(* CoDeSys 2.3.9.59 project: HUS2_AS01_20210128.pro *)
(* Libraries: TcIMX53.lib 21.11.13 13:46:16, TcSUPS_CX9020_U900.lib 4.12.14 20:06:22, STANDARD.LIB 5.6.98 12:03:02, TcBase.lib 14.5.09 12:14:08, TcBaseMath.lib 27.7.04 12:07:56, TcFloatPC.lib 17.3.20 10:16:00, TcHVAC.lib 3.11.16 15:14:26, TcIoFunctions.lib 27.1.17 18:22:22, TcMath.lib 23.9.04 15:15:30, TcPlcCoupler.lib 26.7.12 16:14:58, TcSystem.lib 7.6.16 11:01:22, TcUtilities.lib 3.2.16 17:08:58, TcModbusSrv.lib 11.11.16 10:29:02 *)

(* Task configuration *)
TASK Standard (PRIORITY := 1, INTERVAL := T#20ms);
	MAIN
END_TASK

(* Global variable list: xOvrigt/AcknowledgeFault *)
VAR_GLOBAL
(****************************************************************************************************)
	bReset_Global		AT %Q*:	BOOL;	(*Global reset flag - this flag is common in many programs*)
END_VAR

(* Global variable list: xOvrigt/CtrlVoltage *)
VAR_GLOBAL
	bWithoutMonitoring							:	BOOL:=TRUE;
(*
	bCtrlVoltage_24VAC1		AT%I*			:	BOOL;			(* 24Volt AC1 *)
	bCtrlVoltage_24VAC2		AT%I*			:	BOOL;			(* 24Volt AC2 *)
	bCtrlVoltage_24VAC3		AT%I*			:	BOOL;			(* 24Volt AC3 *)
	bCtrlVoltage_24VAC4		AT%I*			:	BOOL;			(* 24Volt AC4 *)
	bCtrlVoltage_24VAC5		AT%I*			:	BOOL;			(* 24Volt AC5 *)
	bCtrlVoltage_24VAC6		AT%I*			:	BOOL;			(* 24Volt AC6 *)
	bCtrlVoltage_24VAC7		AT%I*			:	BOOL;			(* 24Volt AC7 *)
	bCtrlVoltage_24VAC8		AT%I*			:	BOOL;			(* 24Volt AC8 *)

	bCtrlVoltage_24VDC1	  	AT%I*			:	BOOL;			(* 24Volt DC1 *)
	bCtrlVoltage_24VDC2	  	AT%I*			:	BOOL;			(* 24Volt DC2 *)
	bCtrlVoltage_24VDC3	  	AT%I*			:	BOOL;			(* 24Volt DC3 *)
	bCtrlVoltage_24VDC4	  	AT%I*			:	BOOL;			(* 24Volt DC4 *)
	bCtrlVoltage_24VDC5	  	AT%I*			:	BOOL;			(* 24Volt DC5 *)
	bCtrlVoltage_24VDC6	  	AT%I*			:	BOOL;			(* 24Volt DC6 *)
	bCtrlVoltage_24VDC7	  	AT%I*			:	BOOL;			(* 24Volt DC7 *)
	bCtrlVoltage_24VDC8	  	AT%I*			:	BOOL;			(* 24Volt DC8 *)

	bCtrlVoltage_230VAC1	  	AT%I*			:	BOOL;			(* 230Volt AC1 *)
	bCtrlVoltage_230VAC2		AT%I*			:	BOOL;			(* 230Volt AC2 *)
	bCtrlVoltage_230VAC3	  	AT%I*			:	BOOL;			(* 230Volt AC3 *)
	bCtrlVoltage_230VAC4	  	AT%I*			:	BOOL;			(* 230Volt AC4 *)
	bCtrlVoltage_230VAC5	  	AT%I*			:	BOOL;			(* 230Volt AC5 *)
	bCtrlVoltage_230VAC6	  	AT%I*			:	BOOL;			(* 230Volt AC6 *)
	bCtrlVoltage_230VAC7	  	AT%I*			:	BOOL;			(* 230Volt AC7 *)
	bCtrlVoltage_230VAC8	  	AT%I*			:	BOOL;			(* 230Volt AC8 *)
*)
END_VAR

(* Global variable list: xOvrigt/Globale_Variablen *)
VAR_GLOBAL
	bSetDefault_Global:		BOOL;	(*Global set default flag. This flag is common in many programs*)

END_VAR

(* Global variable list: xOvrigt/GVL *)
VAR_GLOBAL

	HUS2_VV1_GT11_BV	AT%MB3260	:REAL;	(*	HUS2_VV1_GT11_BV	AS01	GVL.HUS2_VV1_GT11_BV	REAL	-50	150	-50	150	°C	0.0	Börvärde framledningstemp tappvarmvatten			*)


END_VAR

(* Global variable list: HUS1/AS02/HUS1_AS02_IO_Hardvara *)
VAR_GLOBAL


										
	(* Digitala in, KL1488  *)									
	(*Kort1*)									
		AS02_Kort01_DI01				AT %I*			:BOOL;	
		AS02_Kort01_DI02				AT %I*			:BOOL;	
		AS02_Kort01_DI03				AT %I*			:BOOL;	
		AS02_Kort01_DI04				AT %I*			:BOOL;	
		AS02_Kort01_DI05				AT %I*			:BOOL;	
		AS02_Kort01_DI06				AT %I*			:BOOL;	
		AS02_Kort01_DI07				AT %I*			:BOOL;	
		AS02_Kort01_DI08				AT %I*			:BOOL;	
										
										
	(* Digitala in, KL1488  *)									
	(*Kort2*)									
		AS02_Kort02_DI01				AT %I*			:BOOL;	
		AS02_Kort02_DI02				AT %I*			:BOOL;	
		AS02_Kort02_DI03				AT %I*			:BOOL;	
		AS02_Kort02_DI04				AT %I*			:BOOL;	
		AS02_Kort02_DI05				AT %I*			:BOOL;	
		AS02_Kort02_DI06				AT %I*			:BOOL;	
		AS02_Kort02_DI07				AT %I*			:BOOL;	
		AS02_Kort02_DI08				AT %I*			:BOOL;	
										
										
	(* Digital Ut, KL2408 *)									
	(*Kort3*)									
		AS02_Kort03_DU01				AT %Q*			:BOOL;	
		AS02_Kort03_DU02				AT %Q*			:BOOL;	
		AS02_Kort03_DU03				AT %Q*			:BOOL;	
		AS02_Kort03_DU04				AT %Q*			:BOOL;	
		AS02_Kort03_DU05				AT %Q*			:BOOL;	
		AS02_Kort03_DU06				AT %Q*			:BOOL;	
		AS02_Kort03_DU07				AT %Q*			:BOOL;	
		AS02_Kort03_DU08				AT %Q*			:BOOL;	
										
										
(*	(* Analoga in, KL3208-0010, PT1000 *)									
	(*Kort5*)									
		AS02_Kort04_AI01								
		AS02_Kort04_AI02								
		AS02_Kort04_AI03								
		AS02_Kort04_AI04								
		AS02_Kort04_AI05								
		AS02_Kort04_AI06								
		AS02_Kort04_AI07								
		AS02_Kort04_AI08					*)			
										

	(* Analoga Ut, KL4408 *)									
	(*Kort5*)									
		AS02_Kort05_AU01				AT %Q*			:INT;	
		AS02_Kort05_AU02				AT %Q*			:INT;	
		AS02_Kort05_AU03				AT %Q*			:INT;	
		AS02_Kort05_AU04				AT %Q*			:INT;	
		AS02_Kort05_AU05				AT %Q*			:INT;	
		AS02_Kort05_AU06				AT %Q*			:INT;	
		AS02_Kort05_AU07				AT %Q*			:INT;	
		AS02_Kort05_AU08				AT %Q*			:INT;	
										
										
										

										
										


END_VAR

(* Global variable list: HUS1/AS02/HUS1_AS02_IO_Program *)
VAR_GLOBAL

					(*	Name	Device	Address	Data type	Rawmin	Rawmax	Engmin	Engmax	Unit	Format	Description	Alarmoptions	Trendoptions	*)	
	(* Digitala in, KL1488  *)																			
	(*Kort 1*)																			
		HUS1_AS02_FB01_L	AT%MX332.0	:BOOL;	(*	HUS1_AS02_FB01_L	AS01	GVL.HUS1_AS02_FB01_L	DIGITAL	0	0	0	0			Fasbrott/fel fasföljd	p:A		*)
		HUS1_AS02_JFB01_L	AT%MX332.1	:BOOL;	(*	HUS1_AS02_JFB01_L	AS01	GVL.HUS1_AS02_JFB01_L	DIGITAL	0	0	0	0			Jordfelsbrytare 	p:B		*)	
		HUS1_AS02_LR01_L	AT%MX332.2	:BOOL;	(*	HUS1_AS02_LR01_L	AS01	GVL.HUS1_AS02_LR01_L	DIGITAL	0	0	0	0			Utlöst dvärgbrytare 	p:B		*)	
		HUS1_AS02_FS01_L	AT%MX332.3	:BOOL;	(*	HUS1_AS02_FS01_L	AS01	GVL.HUS1_AS02_FS01_L	DIGITAL	0	0	0	0			Utlöst finsäkring	p:B		*)	
		HUS1_AS02_RESERV_DI_KORT01_CH05	AT%MX332.4	:BOOL;	(*											Reserv 			*)	
		HUS1_AS02_RESERV_DI_KORT01_CH06	AT%MX332.5	:BOOL;	(*											Reserv 			*)	
		HUS1_AS02_RESERV_DI_KORT01_CH07	AT%MX332.6	:BOOL;	(*											Reserv 			*)	
		HUS1_AS02_RESERV_DI_KORT01_CH08	AT%MX332.7	:BOOL;	(*											Reserv 			*)	
																				

	(* Digitala in, KL1488  *)																			
	(*Kort 2*)																			
		HUS1_VS20_PV01_L	AT%MX333.3	:BOOL;	(*														*)
		HUS1_FA101_FF01_LD	AT%MX333.1	:BOOL;	(*	HUS1_FA101_FF01_LD	AS01	HUS1_AS02_Program.HUS1_FA101_FF01_LD	DIGITAL	0	0	0	0			Driftfel frånluftsfläkt			*)	
		HUS1_FA102_FF01_LD	AT%MX333.2	:BOOL;	(*	HUS1_FA102_FF01_LD	AS01	HUS1_AS02_Program.HUS1_FA102_FF01_LD	DIGITAL	0	0	0	0			Driftfel frånluftsfläkt			*)	
		HUS1_VS20_PV01_IT	AT%MX333.0	:BOOL;	(*	HUS1_VS20_PV01_IT	AS01	HUS1_AS02_Program.HUS1_VS20_PV01_IT	DIGITAL	0	0	0	0			Driftindikering cirkulationspump			*)	
		HUS1_AS02_RESERV_DI_KORT02_CH05	AT%MX333.4	:BOOL;	(*											Reserv 			*)	
		HUS1_AS02_RESERV_DI_KORT02_CH06	AT%MX333.5	:BOOL;	(*											Reserv 			*)	
		HUS1_AS02_RESERV_DI_KORT02_CH07	AT%MX333.6	:BOOL;	(*											Reserv 			*)	
		HUS1_AS02_RESERV_DI_KORT02_CH08	AT%MX333.7	:BOOL;	(*											Reserv 			*)	


	(* Digital Ut, KL2408 *)																			
	(*Kort 3*)																			
		HUS1_AS02_SA01_M	AT%MX334.0	:BOOL;	(*											Summalarm AS01 			*)	
		HUS1_VS20_PV01_M	AT%MX334.1	:BOOL;	(*											Manöver			*)	
		HUS1_AS02_RESERV_DU_KORT03_CH03	AT%MX334.2	:BOOL;	(*											Reserv 			*)	
		HUS1_AS02_RESERV_DU_KORT03_CH04	AT%MX334.3	:BOOL;	(*											Reserv 			*)	
		HUS1_AS02_RESERV_DU_KORT03_CH05	AT%MX334.4	:BOOL;	(*											Reserv 			*)	
		HUS1_AS02_RESERV_DU_KORT03_CH06	AT%MX334.5	:BOOL;	(*											Reserv 			*)	
		HUS1_AS02_RESERV_DU_KORT03_CH07	AT%MX334.6	:BOOL;	(*											Reserv 			*)	
		HUS1_AS02_RESERV_DU_KORT03_CH08	AT%MX334.7	:BOOL;	(*											Reserv 			*)	
																				
																				
	(* Analoga in, KL3208-0010, PT1000  *)																			
	(*Kort 4*)																			
		HUS1_VS20_GT11_MV	AT%MB336	:REAL;	(*	HUS1_VS20_GT11_MV	AS01	GVL.HUS1_VS20_GT11_MV	REAL	-50	150	-50	150	°C	0.0	Mätvärde tilloppstemperatur			*)	
		HUS1_VS20_GT41_MV	AT%MB340	:REAL;	(*	HUS1_VS20_GT41_MV	AS01	GVL.HUS1_VS20_GT41_MV	REAL	-50	150	-50	150	°C	0.0	Mätvärde returtemperatur			*)	
		HUS1_FA101_GT51_MV	AT%MB344	:REAL;	(*	HUS1_FA101_GT51_MV	AS01	GVL.HUS1_FA101_GT51_MV	REAL	-50	150	-50	150	°C	0.0	Mätvärde frånluftstemperatur			*)	
		HUS1_FA102_GT51_MV	AT%MB348	:REAL;	(*	HUS1_FA102_GT51_MV	AS01	GVL.HUS1_FA102_GT51_MV	REAL	-50	150	-50	150	°C	0.0	Mätvärde frånluftstemperatur			*)	
		HUS1_AS02_RESERV_AI_KORT04_CH05	AT%MB352	:REAL;	(*											Reserv			*)	
		HUS1_AS02_RESERV_AI_KORT04_CH06	AT%MB356	:REAL;	(*											Reserv			*)	
		HUS1_AS02_RESERV_AI_KORT04_CH07	AT%MB360	:REAL;	(*											Reserv			*)	
		HUS1_AS02_RESERV_AI_KORT04_CH08	AT%MB364	:REAL;	(*											Reserv			*)	
																				
																				
	(* Analoga ut, KL4408  *)																			
	(*Kort 5*)																			
		HUS1_VS20_SV21_R	AT%MB368	:REAL;	(*	HUS1_VS20_SV21_R	AS01	GVL.HUS1_VS20_SV21_R	REAL	0	100	0	100	%		Styrsignal ventilställdon			*)	
		HUS1_FA101_FF01_R	AT%MB372	:REAL;	(*	HUS1_FA101_FF01_R	AS01	GVL.HUS1_FA101_FF01_R	REAL	0	100	0	100	%		Styrsignal frånluftsfläkt			*)	
		HUS1_FA102_FF01_R	AT%MB376	:REAL;	(*	HUS1_FA102_FF01_R	AS01	GVL.HUS1_FA102_FF01_R	REAL	0	100	0	100	%		Styrsignal frånluftsfläkt			*)	
		HUS1_AS02_RESERV_AU_KORT05_CH04	AT%MB380	:REAL;	(*											Reserv			*)	
		HUS1_AS02_RESERV_AU_KORT05_CH05	AT%MB384	:REAL;	(*											Reserv			*)	
		HUS1_AS02_RESERV_AU_KORT05_CH06	AT%MB388	:REAL;	(*											Reserv			*)	
		HUS1_AS02_RESERV_AU_KORT05_CH07	AT%MB392	:REAL;	(*											Reserv			*)	
		HUS1_AS02_RESERV_AU_KORT05_CH08	AT%MB396	:REAL;	(*											Reserv			*)	
																				
																				
																				
																				

END_VAR

(* Global variable list: HUS1/FA101, FA102/HUS1_FA101_102_INST *)
VAR_GLOBAL PERSISTENT

																			

					(*	Name	Device	Address	Data type	Rawmin	Rawmax	Engmin	Engmax	Unit	Format	Description	Alarmoptions	Trendoptions	*)
																			
		HUS1_FA101_SO1_MAN	AT%MB4600	:INT;	(*	HUS1_FA101_SO1_MAN	AS01	GVL.HUS1_FA101_SO1_MAN	INT	0	2	0	2			Manuell styrning system FA101. 0=Auto, 1=Manuell från, 2=Manuell till			*)
		HUS1_FA101_SO1_FLM	AT%MB4602	:INT;	(*	HUS1_FA101_SO1_FLM	AS01	GVL.HUS1_FA101_SO1_FLM	INT	0	3600	0	3600	Min		Larmfördröjning serviceomkopplare ej i läge AUTO			*)
																			
		HUS1_FA101_FF01_FLM	AT%MB4604	:INT;	(*	HUS1_FA101_FF01_FLM	AS01	GVL.HUS1_FA101_FF01_FLM	INT	0	3600	0	3600	Min		Larmfördröjning frånluftsfläkt ej i AUTO			*)
		HUS1_FA101_FF01_FLD	AT%MB4606	:INT;	(*	HUS1_FA101_FF01_FLD	AS01	GVL.HUS1_FA101_FF01_FLD	INT	0	120	0	120	Sek		Larmfördröjning driftfel frånluftsfläkt			*)
																			
		HUS1_FA101_FF01_MAN	AT%MB4608	:INT;	(*	HUS1_FA101_FF01_MAN	AS01	GVL.HUS1_FA101_FF01_MAN	INT	0	2	0	2			Manuell styrning frånluftsfläkt 0=Auto,1=Från,2=Till			*)
		HUS1_FA101_FF01_MAN1	AT%MB4610	:INT;	(*	HUS1_FA101_FF01_MAN	AS01	GVL.HUS1_FA101_FF01_MAN	INT	0	1	0	1			Manuell styrning styrsignal frånluftsfläkt 0=Auto,1=Till			*)
		HUS1_FA101_FF01_RMAN	AT%MB4612	:REAL;	(*	HUS1_FA101_FF01_RMAN	AS01	GVL.HUS1_FA101_FF01_RMAN	REAL	0	100	0	100	%		Manuell styrsignal frånluftsfläkt			*)
																			
		HUS1_FA101_GT51_STAG	AT%MB4616	:REAL;	(*	HUS1_FA101_GT51_STAG	AS01	GVL.HUS1_FA101_GT51_STAG	REAL	0	50	0	50	°C	0.0	Gränsvärde start forcering frånluftsfläkt			*)
		HUS1_FA101_GT51_STOG	AT%MB4620	:REAL;	(*	HUS1_FA101_GT51_STOG	AS01	GVL.HUS1_FA101_GT51_STOG	REAL	0	50	0	50	°C	0.0	Gränsvärde stopp forcering frånluftsfläkt			*)
																			
		HUS1_FA101_GT51_GVH	AT%MB4624	:REAL;	(*	HUS1_FA101_GT51_GVH	AS01	GVL.HUS1_FA101_GT51_GVH	REAL	0	50	0	50	°C	0.0	Gränsvärde hög temperatur			*)
		HUS1_FA101_GT51_FLG	AT%MB4628	:INT;	(*	HUS1_FA101_GT51_FLG	AS01	GVL.HUS1_FA101_GT51_FLG	INT	0	3600	0	3600	Min		Lamfördröjning hög temperatur			*)
																			
																			
		HUS1_FA101_GT51_KRV	AT%MB4636	:REAL;	(*	HUS1_FA101_GT51_KRV	AS01	GVL.HUS1_FA101_GT51_KRV	REAL	-10	10	-10	10	°C	0.0	Kalibreringsvärde frånluftsgivare			*)
																			
		HUS1_FA101_FF01_BV	AT%MB4640	:REAL;	(*	HUS1_FA101_FF01_BV	AS01	GVL.HUS1_FA101_FF01_BV	REAL	0	100	0	100	%		Grundflöde frånluftsfläkt			*)
		HUS1_FA101_FF01_BV1	AT%MB4644	:REAL;	(*	HUS1_FA101_FF01_BV1	AS01	GVL.HUS1_FA101_FF01_BV1	REAL	0	100	0	100	%		Forcerat flöde frånluftsfläkt			*)
																			
																			
																			
																			
																			
																			
		HUS1_FA102_SO1_MAN	AT%MB4660	:INT;	(*	HUS1_FA102_SO1_MAN	AS01	GVL.HUS1_FA102_SO1_MAN	INT	0	2	0	2			Manuell styrning system FA102. 0=Auto, 1=Manuell från, 2=Manuell till			*)
		HUS1_FA102_SO1_FLM	AT%MB4662	:INT;	(*	HUS1_FA102_SO1_FLM	AS01	GVL.HUS1_FA102_SO1_FLM	INT	0	3600	0	3600	Min		Larmfördröjning serviceomkopplare ej i läge AUTO			*)
																			
		HUS1_FA102_FF01_FLM	AT%MB4664	:INT;	(*	HUS1_FA102_FF01_FLM	AS01	GVL.HUS1_FA102_FF01_FLM	INT	0	3600	0	3600	Min		Larmfördröjning frånluftsfläkt ej i AUTO			*)
		HUS1_FA102_FF01_FLD	AT%MB4666	:INT;	(*	HUS1_FA102_FF01_FLD	AS01	GVL.HUS1_FA102_FF01_FLD	INT	0	120	0	120	Sek		Larmfördröjning driftfel frånluftsfläkt			*)
																			
		HUS1_FA102_FF01_MAN	AT%MB4668	:INT;	(*	HUS1_FA102_FF01_MAN	AS01	GVL.HUS1_FA102_FF01_MAN	INT	0	2	0	2			Manuell styrning frånluftsfläkt 0=Auto,1=Från,2=Till			*)
		HUS1_FA102_FF01_MAN1	AT%MB4670	:INT;	(*	HUS1_FA102_FF01_MAN	AS01	GVL.HUS1_FA102_FF01_MAN	INT	0	1	0	1			Manuell styrning styrsignal frånluftsfläkt 0=Auto,1=Till			*)
		HUS1_FA102_FF01_RMAN	AT%MB4672	:REAL;	(*	HUS1_FA102_FF01_RMAN	AS01	GVL.HUS1_FA102_FF01_RMAN	REAL	0	100	0	100	%		Manuell styrsignal frånluftsfläkt			*)
																			
		HUS1_FA102_GT51_STAG	AT%MB4676	:REAL;	(*	HUS1_FA102_GT51_STAG	AS01	GVL.HUS1_FA102_GT51_STAG	REAL	0	50	0	50	°C	0.0	Gränsvärde start forcering frånluftsfläkt			*)
		HUS1_FA102_GT51_STOG	AT%MB4680	:REAL;	(*	HUS1_FA102_GT51_STOG	AS01	GVL.HUS1_FA102_GT51_STOG	REAL	0	50	0	50	°C	0.0	Gränsvärde stopp forcering frånluftsfläkt			*)
																			
		HUS1_FA102_GT51_GVH	AT%MB4684	:REAL;	(*	HUS1_FA102_GT51_GVH	AS01	GVL.HUS1_FA102_GT51_GVH	REAL	0	50	0	50	°C	0.0	Gränsvärde hög temperatur			*)
		HUS1_FA102_GT51_FLG	AT%MB4688	:INT;	(*	HUS1_FA102_GT51_FLG	AS01	GVL.HUS1_FA102_GT51_FLG	INT	0	3600	0	3600	Min		Lamfördröjning hög temperatur			*)
																			
																			
		HUS1_FA102_GT51_KRV	AT%MB4696	:REAL;	(*	HUS1_FA102_GT51_KRV	AS01	GVL.HUS1_FA102_GT51_KRV	REAL	-10	10	-10	10	°C	0.0	Kalibreringsvärde frånluftsgivare			*)
																			
		HUS1_FA102_FF01_BV	AT%MB4700	:REAL;	(*	HUS1_FA102_FF01_BV	AS01	GVL.HUS1_FA102_FF01_BV	REAL	0	100	0	100	%		Grundflöde frånluftsfläkt			*)
		HUS1_FA102_FF01_BV1	AT%MB4704	:REAL;	(*	HUS1_FA102_FF01_BV1	AS01	GVL.HUS1_FA102_FF01_BV1	REAL	0	100	0	100	%		Forcerat flöde frånluftsfläkt			*)
																			
																			
																			
																			
																			
																			
																			
																			

																			


END_VAR
																
																

(* Global variable list: HUS1/FA101, FA102/HUS1_FA101_102_LARM *)
VAR_GLOBAL



																						
																						
	HUS1_FA101_SO1_LM	AT%MX4780.0	:BOOL; 	(*	HUS1_FA101_SO1_LM	AS01	GVL.HUS1_FA101_SO1_LM	DIGITAL	0	0	0	0			Serviceomkopplare ej i läge AUTO	p:C		*)				
	HUS1_FA101_FF01_LM	AT%MX4780.1	:BOOL; 	(*	HUS1_FA101_FF01_LM	AS01	GVL.HUS1_FA101_FF01_LM	DIGITAL	0	0	0	0			Frånluftsfläkt ej i AUTO	p:B		*)				
	HUS1_FA101_GT51_LG	AT%MX4780.2	:BOOL; 	(*	HUS1_FA101_GT51_LG	AS01	GVL.HUS1_FA101_GT51_LG	DIGITAL	0	0	0	0			Givarfel frånluftsgivare	p:B		*)				
	HUS1_FA101_GT51_LH	AT%MX4780.3	:BOOL; 	(*	HUS1_FA101_GT51_LH	AS01	GVL.HUS1_FA101_GT51_LH	DIGITAL	0	0	0	0			Hög temperatur	p:B		*)				
																						
	HUS1_FA101_FF01_ACK	AT%MX4781.0	:BOOL; 	(*	HUS1_FA101_FF01_ACK	AS01	GVL.HUS1_FA101_FF01_ACK	DIGITAL	0	0	0	0			Larmkvittens frånluftsfläkt			*)				
																						
																						
	HUS1_FA102_SO1_LM	AT%MX4782.0	:BOOL; 	(*	HUS1_FA102_SO1_LM	AS01	GVL.HUS1_FA102_SO1_LM	DIGITAL	0	0	0	0			Serviceomkopplare ej i läge AUTO	p:C		*)				
	HUS1_FA102_FF01_LM	AT%MX4782.1	:BOOL; 	(*	HUS1_FA102_FF01_LM	AS01	GVL.HUS1_FA102_FF01_LM	DIGITAL	0	0	0	0			Frånluftsfläkt ej i AUTO	p:B		*)				
	HUS1_FA102_GT51_LG	AT%MX4782.2	:BOOL; 	(*	HUS1_FA102_GT51_LG	AS01	GVL.HUS1_FA102_GT51_LG	DIGITAL	0	0	0	0			Givarfel frånluftsgivare	p:B		*)				
	HUS1_FA102_GT51_LH	AT%MX4782.3	:BOOL; 	(*	HUS1_FA102_GT51_LH	AS01	GVL.HUS1_FA102_GT51_LH	DIGITAL	0	0	0	0			Hög temperatur	p:B		*)				
																						
	HUS1_FA102_FF01_ACK	AT%MX4784.0	:BOOL; 	(*	HUS1_FA102_FF01_ACK	AS01	GVL.HUS1_FA102_FF01_ACK	DIGITAL	0	0	0	0			Larmkvittens frånluftsfläkt			*)				
																						
																						
																						
																						



END_VAR

(* Global variable list: HUS1/FA101, FA102/HUS1_FA101_102_OVRIGT *)
VAR_GLOBAL


																				
	HUS1_FA101_SO1_IH	AT%MX4900.0	:BOOL;	(*	HUS1_FA101_SO1_IH	AS01	GVL.HUS1_FA101_SO1_IH	DIGITAL	0	0	0	0			Serviceomkopplare ej i AUTO			*)		
	HUS1_FA101_SO1_IA	AT%MX4900.1	:BOOL;	(*	HUS1_FA101_SO1_IA	AS01	GVL.HUS1_FA101_SO1_IA	DIGITAL	0	0	0	0			Serviceomkopplare i läge AUTO			*)		
	HUS1_FA101_SO1_IF	AT%MX4900.2	:BOOL;	(*	HUS1_FA101_SO1_IF	AS01	GVL.HUS1_FA101_SO1_IF	DIGITAL	0	0	0	0			Serviceomkopplare i läge 0			*)		
	HUS1_FA101_SO1_IT	AT%MX4900.3	:BOOL;	(*	HUS1_FA101_SO1_IT	AS01	GVL.HUS1_FA101_SO1_IT	DIGITAL	0	0	0	0			Serviceomkopplare i läge HAND TILL			*)		
																				
	HUS1_FA101_FF01_IT	AT%MX4900.5	:BOOL;	(*	HUS1_FA101_FF01_IT	AS01	GVL.HUS1_FA101_FF01_IT	DIGITAL	0	0	0	0			Frånluftsfläkt indikering TILL			*)		
																				
																				
	HUS1_FA102_SO1_IH	AT%MX4901.0	:BOOL;	(*	HUS1_FA102_SO1_IH	AS01	GVL.HUS1_FA102_SO1_IH	DIGITAL	0	0	0	0			Serviceomkopplare ej i AUTO			*)		
	HUS1_FA102_SO1_IA	AT%MX4901.1	:BOOL;	(*	HUS1_FA102_SO1_IA	AS01	GVL.HUS1_FA102_SO1_IA	DIGITAL	0	0	0	0			Serviceomkopplare i läge AUTO			*)		
	HUS1_FA102_SO1_IF	AT%MX4901.2	:BOOL;	(*	HUS1_FA102_SO1_IF	AS01	GVL.HUS1_FA102_SO1_IF	DIGITAL	0	0	0	0			Serviceomkopplare i läge 0			*)		
	HUS1_FA102_SO1_IT	AT%MX4901.3	:BOOL;	(*	HUS1_FA102_SO1_IT	AS01	GVL.HUS1_FA102_SO1_IT	DIGITAL	0	0	0	0			Serviceomkopplare i läge HAND TILL			*)		
																				
	HUS1_FA102_FF01_IT	AT%MX4901.5	:BOOL;	(*	HUS1_FA102_FF01_IT	AS01	GVL.HUS1_FA102_FF01_IT	DIGITAL	0	0	0	0			Frånluftsfläkt indikering TILL			*)		
																				
																				
																				
																				



END_VAR

(* Global variable list: HUS1/VS20/HUS1_VS20_INST *)
VAR_GLOBAL PERSISTENT


																			
					(*	Name	Device	Address	Data type	Rawmin	Rawmax	Engmin	Engmax	Unit	Format	Description	Alarmoptions	Trendoptions	*)
																			
		HUS1_VS20_GT11_UX1	AT%MB4392	:REAL;	(*	HUS1_VS20_GT11_UX1	AS01	GVL.HUS1_VS20_GT11_UX1	REAL	-50	150	-50	150	°C	0.0	Utetemp. kompenserad kurva Brytpunkt X1			*)
		HUS1_VS20_GT11_UX2	AT%MB4396	:REAL;	(*	HUS1_VS20_GT11_UX2	AS01	GVL.HUS1_VS20_GT11_UX2	REAL	-50	150	-50	150	°C	0.0	Utetemp. kompenserad kurva Brytpunkt X2			*)
		HUS1_VS20_GT11_UX3	AT%MB4400	:REAL;	(*	HUS1_VS20_GT11_UX3	AS01	GVL.HUS1_VS20_GT11_UX3	REAL	-50	150	-50	150	°C	0.0	Utetemp. kompenserad kurva Brytpunkt X3			*)
		HUS1_VS20_GT11_UX4	AT%MB4404	:REAL;	(*	HUS1_VS20_GT11_UX4	AS01	GVL.HUS1_VS20_GT11_UX4	REAL	-50	150	-50	150	°C	0.0	Utetemp. kompenserad kurva Brytpunkt X4			*)
		HUS1_VS20_GT11_UX5	AT%MB4408	:REAL;	(*	HUS1_VS20_GT11_UX5	AS01	GVL.HUS1_VS20_GT11_UX5	REAL	-50	150	-50	150	°C	0.0	Utetemp. kompenserad kurva Brytpunkt X5			*)
		HUS1_VS20_GT11_UY1	AT%MB4412	:REAL;	(*	HUS1_VS20_GT11_UY1	AS01	GVL.HUS1_VS20_GT11_UY1	REAL	0	150	0	150	°C	0.0	Utetemp. kompenserad kurva Brytpunkt Y1			*)
		HUS1_VS20_GT11_UY2	AT%MB4416	:REAL;	(*	HUS1_VS20_GT11_UY2	AS01	GVL.HUS1_VS20_GT11_UY2	REAL	0	150	0	150	°C	0.0	Utetemp. kompenserad kurva Brytpunkt Y2			*)
		HUS1_VS20_GT11_UY3	AT%MB4420	:REAL;	(*	HUS1_VS20_GT11_UY3	AS01	GVL.HUS1_VS20_GT11_UY3	REAL	0	150	0	150	°C	0.0	Utetemp. kompenserad kurva Brytpunkt Y3			*)
		HUS1_VS20_GT11_UY4	AT%MB4424	:REAL;	(*	HUS1_VS20_GT11_UY4	AS01	GVL.HUS1_VS20_GT11_UY4	REAL	0	150	0	150	°C	0.0	Utetemp. kompenserad kurva Brytpunkt Y4			*)
		HUS1_VS20_GT11_UY5	AT%MB4428	:REAL;	(*	HUS1_VS20_GT11_UY5	AS01	GVL.HUS1_VS20_GT11_UY5	REAL	0	150	0	150	°C	0.0	Utetemp. kompenserad kurva Brytpunkt Y5			*)
		HUS1_VS20_GT11_UMIN	AT%MB4432	:REAL;	(*	HUS1_VS20_GT11_UMIN	AS01	GVL.HUS1_VS20_GT11_UMIN	REAL	0	150	0	150	°C	0.0	Utetemp. kompenserad kurva Min-begränsning			*)
		HUS1_VS20_GT11_UMAX	AT%MB4436	:REAL;	(*	HUS1_VS20_GT11_UMAX	AS01	GVL.HUS1_VS20_GT11_UMAX	REAL	0	150	0	150	°C	0.0	Utetemp. kompenserad kurva Max-begränsning			*)
																			
		HUS1_VS20_GT11_CP	AT%MB4440	:REAL;	(*	HUS1_VS20_GT11_CPV	AS01	GVL.HUS1_VS20_GT11_CP	REAL	0	10	0	10		0.0	P-parameter			*)
		HUS1_VS20_GT11_CI	AT%MB4444	:REAL;	(*	HUS1_VS20_GT11_CIV	AS01	GVL.HUS1_VS20_GT11_CI	REAL	0	900	0	900	Sek		I-Tid 			*)
		HUS1_VS20_GT11_CD	AT%MB4448	:REAL;	(*	HUS1_VS20_GT11_CDV	AS01	GVL.HUS1_VS20_GT11_CD	REAL	0	900	0	900	Sek		D-tid 			*)
		HUS1_VS20_GT11_CS	AT%MB4452	:REAL;	(*	HUS1_VS20_GT11_CSV	AS01	GVL.HUS1_VS20_GT11_CS	REAL	0	900	0	900	Sek		Samplingstid			*)
		HUS1_VS20_GT11_CZ	AT%MB4456	:REAL;	(*	HUS1_VS20_GT11_CZV	AS01	GVL.HUS1_VS20_GT11_CZ	REAL	-10	10	-10	10	°C	0.0	Dödband regulator			*)
																			
		HUS1_VS20_SO1_MAN	AT%MB4460	:INT;	(*	HUS1_VS20_SO1_MAN	AS01	GVL.HUS1_VS20_SO1_MAN	INT	0	2	0	2			Manuell styrning system VS20. 0=Auto, 1=Manuell från, 2=Manuell till			*)
		HUS1_VS20_PV01_MAN	AT%MB4462	:INT;	(*	HUS1_VS20_PV01_MAN	AS01	GVL.HUS1_VS20_PV01_MAN	INT	0	2	0	2			Manuell styrning crikulationspump 0=Auto,1=Från,2=Till			*)
		HUS1_VS20_SV21_MAN1	AT%MB4464	:INT;	(*	HUS1_VS20_SV21_MAN	AS01	GVL.HUS1_VS20_SV21_MAN	INT	0	1	0	1			Manuell styrning ventilställdon 0=Auto,1=Hand			*)
		HUS1_VS20_SV21_RMAN	AT%MB4468	:REAL;	(*	HUS1_VS20_SV21_RMAN	AS01	GVL.HUS1_VS20_SV21_RMAN	REAL	0	100	0	100	%		Manuell styrsignal ventilställdon			*)
																			
		HUS1_VS20_SO1_FLM	AT%MB4472	:INT;	(*	HUS1_VS20_SO1_FLM	AS01	GVL.HUS1_VS20_SO1_FLM	INT	0	3600	0	3600	Min		Larmfördröjning serviceomkopplare ej i läge AUTO			*)
		HUS1_VS20_PV01_FLM	AT%MB4474	:INT;	(*	HUS1_VS20_PV01_FLM	AS01	GVL.HUS1_VS20_PV01_FLM	INT	0	3600	0	3600	Min		Larmfördröjning cirkulationspump ej i AUTO			*)
		HUS1_VS20_SV21_FLM	AT%MB4476	:INT;	(*	HUS1_VS20_SV21_FLM	AS01	GVL.HUS1_VS20_SV21_FLM	INT	0	3600	0	3600	Min		Larmfördröjning ventilställdon ej i AUTO			*)
		HUS1_VS20_PV01_FLD	AT%MB4478	:INT;	(*	HUS1_VS20_PV01_FLD	AS01	GVL.HUS1_VS20_PV01_FLD	INT	0	120	0	120	Sek		Larmfördröjning driftfel cirkulationspump			*)
																			
		HUS1_VS20_GT11_GAVH	AT%MB4484	:REAL;	(*	HUS1_VS20_GT11_GAVH	AS01	GVL.HUS1_VS20_GT11_GAVH	REAL	-20	20	-20	20	°C	0.0	Gränsavvikelse hög framledningstemperatur			*)
		HUS1_VS20_GT11_GAVL	AT%MB4488	:REAL;	(*	HUS1_VS20_GT11_GAVL	AS01	GVL.HUS1_VS20_GT11_GAVL	REAL	-20	20	-20	20	°C	0.0	Gränsavvikelse låg framledningstemperatur			*)
		HUS1_VS20_GT11_FLAH	AT%MB4492	:INT;	(*	HUS1_VS20_GT11_FLAH	AS01	GVL.HUS1_VS20_GT11_FLAH	INT	0	3600	0	3600	Min		Larmfördröjning hög framledningstemperatur			*)
		HUS1_VS20_GT11_FLAL	AT%MB4494	:INT;	(*	HUS1_VS20_GT11_FLAL	AS01	GVL.HUS1_VS20_GT11_FLAL	INT	0	3600	0	3600	Min		Lamfördröjning låg framledningstemperatur			*)
																			
																			
																			
																			
																			
																			
																			
																			
																			
		HUS1_VS20_GT11_KRV	AT%MB4496	:REAL;	(*	HUS1_VS20_GT11_KRV	AS01	GVL.HUS1_VS20_GT11_KRV	REAL	-10	10	-10	10	°C	0.0	Kalibreringsvärde framledningsgivare			*)
		HUS1_VS20_GT41_KRV	AT%MB4500	:REAL;	(*	HUS1_VS20_GT41_KRV	AS01	GVL.HUS1_VS20_GT41_KRV	REAL	-10	10	-10	10	°C	0.0	Kalibreringsvärde returgivare			*)
																			
																			
																			
		HUS1_VS20_GT11_X1	AT%MB4504	:REAL;	(*	HUS1_VS20_GT11_X1	AS01	GVL.HUS1_VS20_GT11_X1	REAL	-50	150	-50	150	°C	0.0	Effektbegränsning kurva Brytpunkt X1			*)
		HUS1_VS20_GT11_X2	AT%MB4508	:REAL;	(*	HUS1_VS20_GT11_X2	AS01	GVL.HUS1_VS20_GT11_X2	REAL	-50	150	-50	150	°C	0.0	Effektbegränsning kurva Brytpunkt X2			*)
		HUS1_VS20_GT11_X3	AT%MB4512	:REAL;	(*	HUS1_VS20_GT11_X3	AS01	GVL.HUS1_VS20_GT11_X3	REAL	-50	150	-50	150	°C	0.0	Effektbegränsning kurva Brytpunkt X3			*)
		HUS1_VS20_GT11_X4	AT%MB4516	:REAL;	(*	HUS1_VS20_GT11_X4	AS01	GVL.HUS1_VS20_GT11_X4	REAL	-50	150	-50	150	°C	0.0	Effektbegränsning kurva Brytpunkt X4			*)
		HUS1_VS20_GT11_X5	AT%MB4520	:REAL;	(*	HUS1_VS20_GT11_X5	AS01	GVL.HUS1_VS20_GT11_X5	REAL	-50	150	-50	150	°C	0.0	Effektbegränsning kurva Brytpunkt X5			*)
		HUS1_VS20_GT11_Y1	AT%MB4524	:REAL;	(*	HUS1_VS20_GT11_Y1	AS01	GVL.HUS1_VS20_GT11_Y1	REAL	0	150	0	150	°C	0.0	Effektbegränsning kurva Brytpunkt Y1			*)
		HUS1_VS20_GT11_Y2	AT%MB4528	:REAL;	(*	HUS1_VS20_GT11_Y2	AS01	GVL.HUS1_VS20_GT11_Y2	REAL	0	150	0	150	°C	0.0	Effektbegränsning kurva Brytpunkt Y2			*)
		HUS1_VS20_GT11_Y3	AT%MB4532	:REAL;	(*	HUS1_VS20_GT11_Y3	AS01	GVL.HUS1_VS20_GT11_Y3	REAL	0	150	0	150	°C	0.0	Effektbegränsning kurva Brytpunkt Y3			*)
		HUS1_VS20_GT11_Y4	AT%MB4536	:REAL;	(*	HUS1_VS20_GT11_Y4	AS01	GVL.HUS1_VS20_GT11_Y4	REAL	0	150	0	150	°C	0.0	Effektbegränsning kurva Brytpunkt Y4			*)
		HUS1_VS20_GT11_Y5	AT%MB4540	:REAL;	(*	HUS1_VS20_GT11_Y5	AS01	GVL.HUS1_VS20_GT11_Y5	REAL	0	150	0	150	°C	0.0	Effektbegränsning kurva Brytpunkt Y5			*)
		HUS1_VS20_GT11_MIN	AT%MB4544	:REAL;	(*	HUS1_VS20_GT11_MIN	AS01	GVL.HUS1_VS20_GT11_MIN	REAL	0	150	0	150	°C	0.0	Effektbegränsning kurva Min-begränsning			*)
		HUS1_VS20_GT11_MAX	AT%MB4548	:REAL;	(*	HUS1_VS20_GT11_MAX	AS01	GVL.HUS1_VS20_GT11_MAX	REAL	0	150	0	150	°C	0.0	Effektbegränsning kurva Max-begränsning			*)
																			
																			
																			
																			
																			
																			
																			



END_VAR
																
																

(* Global variable list: HUS1/VS20/HUS1_VS20_LARM *)
VAR_GLOBAL


																				
																				
		HUS1_VS20_SO1_LM	AT%MX4570.0	:BOOL; 	(*	HUS1_VS20_SO1_LM	AS01	GVL.HUS1_VS20_SO1_LM	DIGITAL	0	0	0	0			Serviceomkopplare ej i läge AUTO	p:C		*)	
		HUS1_VS20_PV01_LM	AT%MX4570.1	:BOOL; 	(*	HUS1_VS20_PV01_LM	AS01	GVL.HUS1_VS20_PV01_LM	DIGITAL	0	0	0	0			Cirkulationspump ej i AUTO	p:B		*)	
		HUS1_VS20_SV21_LM	AT%MX4570.2	:BOOL; 	(*	HUS1_VS20_SV21_LM	AS01	GVL.HUS1_VS20_SV21_LM	DIGITAL	0	0	0	0			Ventilställdon ej i AUTO	p:B		*)	
		HUS1_VS20_PV01_LD	AT%MX4570.3	:BOOL; 	(*	HUS1_VS20_PV01_LD	AS01	GVL.HUS1_VS20_PV01_LD	DIGITAL	0	0	0	0			Driftfel cirkulationspump	p:B		*)	
		HUS1_VS20_GT11_LG	AT%MX4570.4	:BOOL; 	(*	HUS1_VS20_GT11_LG	AS01	GVL.HUS1_VS20_GT11_LG	DIGITAL	0	0	0	0			Givarfel framledningsgivare	p:B		*)	
		HUS1_VS20_GT41_LG	AT%MX4570.5	:BOOL; 	(*	HUS1_VS20_GT41_LG	AS01	GVL.HUS1_VS20_GT41_LG	DIGITAL	0	0	0	0			Givarfel returgivare	p:B		*)	
		HUS1_VS20_GT11_LAH	AT%MX4570.6	:BOOL; 	(*	HUS1_VS20_GT11_LAH	AS01	GVL.HUS1_VS20_GT11_LAH	DIGITAL	0	0	0	0			Larmavvikelse hög framledningstemp	p:B		*)	
		HUS1_VS20_GT11_LAL	AT%MX4570.7	:BOOL; 	(*	HUS1_VS20_GT11_LAL	AS01	GVL.HUS1_VS20_GT11_LAL	DIGITAL	0	0	0	0			Larmavvikelse låg framledningstemp	p:B		*)	
																				
																				
																				
																				
																				
																				
																				
																				
																				
																				
																				
		HUS1_VS20_PV01_ACK	AT%MX4573.0	:BOOL; 	(*	HUS1_VS20_PV01_ACK	AS01	GVL.HUS1_VS20_PV01_ACK	DIGITAL	0	0	0	0			Larmkvittens pump			*)	
																				
																				
																				
																				
																				
																				


END_VAR

(* Global variable list: HUS1/VS20/HUS1_VS20_OVRIGT *)
VAR_GLOBAL


																						
	HUS1_VS20_SO1_IH	AT%MX4575.0	:BOOL;	(*	HUS1_VS20_SO1_IH	AS01	GVL.HUS1_VS20_SO1_IH	DIGITAL	0	0	0	0			Serviceomkopplare ej i AUTO			*)				
	HUS1_VS20_SO1_IA	AT%MX4575.1	:BOOL;	(*	HUS1_VS20_SO1_IA	AS01	GVL.HUS1_VS20_SO1_IA	DIGITAL	0	0	0	0			Serviceomkopplare i läge AUTO			*)				
	HUS1_VS20_SO1_IF	AT%MX4575.2	:BOOL;	(*	HUS1_VS20_SO1_IF	AS01	GVL.HUS1_VS20_SO1_IF	DIGITAL	0	0	0	0			Serviceomkopplare i läge 0			*)				
	HUS1_VS20_SO1_IT	AT%MX4575.3	:BOOL;	(*	HUS1_VS20_SO1_IT	AS01	GVL.HUS1_VS20_SO1_IT	DIGITAL	0	0	0	0			Serviceomkopplare i läge HAND TILL			*)				
																						
																						
																						
																						
																						
																						
																						
																						
																						
																						
																						
																						
	HUS1_VS20_GT11_BB	AT%MB4576	:REAL;	(*	HUS1_VS20_GT11_BB	AS01	GVL.HUS1_VS20_GT11_BB	REAL	0	150	0	150	°C	0.0	Beräknat börvärde framledningstemperatur			*)				
	HUS1_VS20_GT11_BB1	AT%MB4580	:REAL;	(*	HUS1_VS20_GT11_BB1	AS01	GVL.HUS1_VS20_GT11_BB1	REAL	0	150	0	150	°C	0.0	Beräknad förskjutning framledningstemperatur			*)				
																						
																						
																						
																						
																						


																					

END_VAR

(* Global variable list: HUS2/AL01/HUS2_AL01_IO_Hardvara *)
VAR_GLOBAL


	(* Digitala in, KL1488  *)									
	(*Kort1*)									
		AL01_Kort01_DI01				AT %I*			:BOOL;	
		AL01_Kort01_DI02				AT %I*			:BOOL;	
		AL01_Kort01_DI03				AT %I*			:BOOL;	
		AL01_Kort01_DI04				AT %I*			:BOOL;	
		AL01_Kort01_DI05				AT %I*			:BOOL;	
		AL01_Kort01_DI06				AT %I*			:BOOL;	
		AL01_Kort01_DI07				AT %I*			:BOOL;	
		AL01_Kort01_DI08				AT %I*			:BOOL;	
										
										
	(* Digitala in, KL1488  *)									
	(*Kort2*)									
		AL01_Kort02_DI01				AT %I*			:BOOL;	
		AL01_Kort02_DI02				AT %I*			:BOOL;	
		AL01_Kort02_DI03				AT %I*			:BOOL;	
		AL01_Kort02_DI04				AT %I*			:BOOL;	
		AL01_Kort02_DI05				AT %I*			:BOOL;	
		AL01_Kort02_DI06				AT %I*			:BOOL;	
		AL01_Kort02_DI07				AT %I*			:BOOL;	
		AL01_Kort02_DI08				AT %I*			:BOOL;	
										
										
	(* Digital Ut, KL2408 *)									
	(*Kort3*)									
		AL01_Kort03_DU01				AT %Q*			:BOOL;
		AL01_Kort03_DU02				AT %Q*			:BOOL;	
		AL01_Kort03_DU03				AT %Q*			:BOOL;	
		AL01_Kort03_DU04				AT %Q*			:BOOL;	
		AL01_Kort03_DU05				AT %Q*			:BOOL;	
		AL01_Kort03_DU06				AT %Q*			:BOOL;	
		AL01_Kort03_DU07				AT %Q*			:BOOL;	
		AL01_Kort03_DU08				AT %Q*			:BOOL;	
										
										

												

END_VAR

(* Global variable list: HUS2/AL01/HUS2_AL01_IO_Program *)
VAR_GLOBAL



					(*	Name	Device	Address	Data type	Rawmin	Rawmax	Engmin	Engmax	Unit	Format	Description	Alarmoptions	Trendoptions	*)
	(* Digitala in, KL1488  *)																			
	(*Kort 1*)																			
		HUS2_AL01_FS01_L	AT%MX220.0	:BOOL;	(*	HUS2_AL01_FS01_L	AS01	GVL.HUS2_AL01_FS01_L	DIGITAL	0	0	0	0			Utlöst dvärgbrytare 	p:B		*)	
		HUS2_LB03_HD72_L	AT%MX220.1	:BOOL;	(*	HUS2_LB03_HD72_L	AS01	GVL.HUS2_LB03_HD72_L	DIGITAL	0	0	0	0			Utlöst rökdetektor 	p:A		*)	
		HUS2_LB03_HD72_L1	AT%MX220.2	:BOOL;	(*	HUS2_LB03_HD72_L1	AS01	GVL.HUS2_LB03_HD72_L1	DIGITAL	0	0	0	0			Servicelarm	p:B		*)	
		HUS2_LB03_HD72_L2	AT%MX220.3	:BOOL;	(*	HUS2_LB03_HD72_L2	AS01	GVL.HUS2_LB03_HD72_L2	DIGITAL	0	0	0	0			Fellarm 	p:B		*)	
		HUS2_LB03_BS201_IO	AT%MX220.4	:BOOL;	(*	HUS2_LB03_BS201_IO	AS01	GVL.HUS2_LB03_BS201_IO	DIGITAL	0	0	0	0			Indikering öppet 			*)	
		HUS2_LB03_BS201_IS	AT%MX220.5	:BOOL;	(*	HUS2_LB03_BS201_IS	AS01	GVL.HUS2_LB03_BS201_IS	DIGITAL	0	0	0	0			Indikering stängt 			*)	
		HUS2_LB03_BS202_IO	AT%MX220.6	:BOOL;	(*	HUS2_LB03_BS202_IO	AS01	GVL.HUS2_LB03_BS202_IO	DIGITAL	0	0	0	0			Indikering öppet 			*)	
		HUS2_LB03_BS202_IS	AT%MX220.7	:BOOL;	(*	HUS2_LB03_BS202_IS	AS01	GVL.HUS2_LB03_BS202_IS	DIGITAL	0	0	0	0			Indikering stängt 			*)	
																				
																				
	(* Digitala in, KL1488  *)																			
	(*Kort 2*)																			
		HUS2_LB03_HD71_L	AT%MX221.0	:BOOL;	(*	HUS2_LB03_HD71_L	AS01	GVL.HUS2_LB03_HD71_L	DIGITAL	0	0	0	0			Utlöst rökdetektor 	p:A		*)	
		HUS2_LB03_HD71_L1	AT%MX221.1	:BOOL;	(*	HUS2_LB03_HD71_L1	AS01	GVL.HUS2_LB03_HD71_L1	DIGITAL	0	0	0	0			Servicelarm	p:B		*)	
		HUS2_LB03_HD71_L2	AT%MX221.2	:BOOL;	(*	HUS2_LB03_HD71_L2	AS01	GVL.HUS2_LB03_HD71_L2	DIGITAL	0	0	0	0			Fellarm 	p:B		*)	
		HUS2_LB03_BS203_IO	AT%MX221.3	:BOOL;	(*	HUS2_LB03_BS203_IO	AS01	GVL.HUS2_LB03_BS203_IO	DIGITAL	0	0	0	0			Indikering öppet 			*)	
		HUS2_LB03_BS203_IS	AT%MX221.4	:BOOL;	(*	HUS2_LB03_BS203_IS	AS01	GVL.HUS2_LB03_BS203_IS	DIGITAL	0	0	0	0			Indikering stängt 			*)	
		HUS2_AL01_RESERV_DI_KORT02_CH06	AT%MX221.5	:BOOL;	(*											Reserv 			*)	
		HUS2_AL01_RESERV_DI_KORT02_CH07	AT%MX221.6	:BOOL;	(*											Reserv 			*)	
		HUS2_AL01_RESERV_DI_KORT02_CH08	AT%MX221.7	:BOOL;	(*											Reserv 			*)	
																				
																				
	(* Digital Ut, KL2408 *)																			
	(*Kort 3*)																			
		HUS2_LB03_BS201_M	AT%MX222.0	:BOOL;	(*											Manöver			*)	
		HUS2_LB03_BS202_M	AT%MX222.1	:BOOL;	(*											Manöver			*)	
		HUS2_LB03_BS203_M	AT%MX222.2	:BOOL;	(*											Manöver 			*)	
		HUS2_AL01_RESERV_DU_KORT03_CH04	AT%MX222.3	:BOOL;	(*											Reserv 			*)	
		HUS2_AL01_RESERV_DU_KORT03_CH05	AT%MX222.4	:BOOL;	(*											Reserv 			*)	
		HUS2_AL01_RESERV_DU_KORT03_CH06	AT%MX222.5	:BOOL;	(*											Reserv 			*)	
		HUS2_AL01_RESERV_DU_KORT03_CH07	AT%MX222.6	:BOOL;	(*											Reserv 			*)	
		HUS2_AL01_RESERV_DU_KORT03_CH08	AT%MX222.7	:BOOL;	(*											Reserv 			*)	
																				
																				


END_VAR

(* Global variable list: HUS2/AS01/HUS2_AS01_INST *)
VAR_GLOBAL PERSISTENT

																				
					(*	Name	Device	Address	Data type	Rawmin	Rawmax	Engmin	Engmax	Unit	Format	Description	Alarmoptions	Trendoptions	*)	
	(* Tidkanal belysning fasad *)																			
		HUS2_AS01_BE01_CT1	AT%MB1100	:INT;	(*	HUS2_AS01_BE01_CT1	AS01	GVL.HUS2_AS01_BE01_CT1	INT	0	2359	0	2359	HHMM		Tidkanal BE01 Tillslag 1 Måndag			*)
		HUS2_AS01_BE01_CT2	AT%MB1102	:INT;	(*	HUS2_AS01_BE01_CT2	AS01	GVL.HUS2_AS01_BE01_CT2	INT	0	2359	0	2359	HHMM		Tidkanal BE01 Tillslag 1 Tisdag			*)	
		HUS2_AS01_BE01_CT3	AT%MB1104	:INT;	(*	HUS2_AS01_BE01_CT3	AS01	GVL.HUS2_AS01_BE01_CT3	INT	0	2359	0	2359	HHMM		Tidkanal BE01 Tillslag 1 Onsdag			*)	
		HUS2_AS01_BE01_CT4	AT%MB1106	:INT;	(*	HUS2_AS01_BE01_CT4	AS01	GVL.HUS2_AS01_BE01_CT4	INT	0	2359	0	2359	HHMM		Tidkanal BE01 Tillslag 1 Torsdag			*)	
		HUS2_AS01_BE01_CT5	AT%MB1108	:INT;	(*	HUS2_AS01_BE01_CT5	AS01	GVL.HUS2_AS01_BE01_CT5	INT	0	2359	0	2359	HHMM		Tidkanal BE01 Tillslag 1 Fredag			*)	
		HUS2_AS01_BE01_CT6	AT%MB1110	:INT;	(*	HUS2_AS01_BE01_CT6	AS01	GVL.HUS2_AS01_BE01_CT6	INT	0	2359	0	2359	HHMM		Tidkanal BE01 Tillslag 1 Lördag			*)
		HUS2_AS01_BE01_CT7	AT%MB1112	:INT;	(*	HUS2_AS01_BE01_CT7	AS01	GVL.HUS2_AS01_BE01_CT7	INT	0	2359	0	2359	HHMM		Tidkanal BE01 Tillslag 1 Söndag			*)	
		HUS2_AS01_BE01_CT8	AT%MB1114	:INT;	(*	HUS2_AS01_BE01_CT8	AS01	GVL.HUS2_AS01_BE01_CT8	INT	0	2359	0	2359	HHMM		Tidkanal BE01 Tillslag 1 Helgafton			*)	
		HUS2_AS01_BE01_CT9	AT%MB1116	:INT;	(*	HUS2_AS01_BE01_CT9	AS01	GVL.HUS2_AS01_BE01_CT9	INT	0	2359	0	2359	HHMM		Tidkanal BE01 Tillslag 1 Helgdag			*)	
		HUS2_AS01_BE01_CT11	AT%MB1118	:INT;	(*	HUS2_AS01_BE01_CT11	AS01	GVL.HUS2_AS01_BE01_CT11	INT	0	2359	0	2359	HHMM		Tidkanal BE01 Tillslag 2 Måndag			*)	
		HUS2_AS01_BE01_CT12	AT%MB1120	:INT;	(*	HUS2_AS01_BE01_CT12	AS01	GVL.HUS2_AS01_BE01_CT12	INT	0	2359	0	2359	HHMM		Tidkanal BE01 Tillslag 2 Tisdag			*)	
		HUS2_AS01_BE01_CT13	AT%MB1122	:INT;	(*	HUS2_AS01_BE01_CT13	AS01	GVL.HUS2_AS01_BE01_CT13	INT	0	2359	0	2359	HHMM		Tidkanal BE01 Tillslag 2 Onsdag			*)	
		HUS2_AS01_BE01_CT14	AT%MB1124	:INT;	(*	HUS2_AS01_BE01_CT14	AS01	GVL.HUS2_AS01_BE01_CT14	INT	0	2359	0	2359	HHMM		Tidkanal BE01 Tillslag 2 Torsdag			*)	
		HUS2_AS01_BE01_CT15	AT%MB1126	:INT;	(*	HUS2_AS01_BE01_CT15	AS01	GVL.HUS2_AS01_BE01_CT15	INT	0	2359	0	2359	HHMM		Tidkanal BE01 Tillslag 2 Fredag			*)	
		HUS2_AS01_BE01_CT16	AT%MB1128	:INT;	(*	HUS2_AS01_BE01_CT16	AS01	GVL.HUS2_AS01_BE01_CT16	INT	0	2359	0	2359	HHMM		Tidkanal BE01 Tillslag 2 Lördag			*)	
		HUS2_AS01_BE01_CT17	AT%MB1130	:INT;	(*	HUS2_AS01_BE01_CT17	AS01	GVL.HUS2_AS01_BE01_CT17	INT	0	2359	0	2359	HHMM		Tidkanal BE01 Tillslag 2 Söndag			*)	
		HUS2_AS01_BE01_CT18	AT%MB1132	:INT;	(*	HUS2_AS01_BE01_CT18	AS01	GVL.HUS2_AS01_BE01_CT18	INT	0	2359	0	2359	HHMM		Tidkanal BE01 Tillslag 2 Helgafton			*)	
		HUS2_AS01_BE01_CT19	AT%MB1134	:INT;	(*	HUS2_AS01_BE01_CT19	AS01	GVL.HUS2_AS01_BE01_CT19	INT	0	2359	0	2359	HHMM		Tidkanal BE01 Tillslag 2 Helgdag			*)	
		HUS2_AS01_BE01_CF1	AT%MB1136	:INT;	(*	HUS2_AS01_BE01_CF1	AS01	GVL.HUS2_AS01_BE01_CF1	INT	0	2359	0	2359	HHMM		Tidkanal BE01 Frånslag 1 Måndag			*)	
		HUS2_AS01_BE01_CF2	AT%MB1138	:INT;	(*	HUS2_AS01_BE01_CF2	AS01	GVL.HUS2_AS01_BE01_CF2	INT	0	2359	0	2359	HHMM		Tidkanal BE01 Frånslag 1 Tisdag			*)	
		HUS2_AS01_BE01_CF3	AT%MB1140	:INT;	(*	HUS2_AS01_BE01_CF3	AS01	GVL.HUS2_AS01_BE01_CF3	INT	0	2359	0	2359	HHMM		Tidkanal BE01 Frånslag 1 Onsdag			*)	
		HUS2_AS01_BE01_CF4	AT%MB1142	:INT;	(*	HUS2_AS01_BE01_CF4	AS01	GVL.HUS2_AS01_BE01_CF4	INT	0	2359	0	2359	HHMM		Tidkanal BE01 Frånslag 1 Torsdag			*)	
		HUS2_AS01_BE01_CF5	AT%MB1144	:INT;	(*	HUS2_AS01_BE01_CF5	AS01	GVL.HUS2_AS01_BE01_CF5	INT	0	2359	0	2359	HHMM		Tidkanal BE01 Frånslag 1 Fredag			*)	
		HUS2_AS01_BE01_CF6	AT%MB1146	:INT;	(*	HUS2_AS01_BE01_CF6	AS01	GVL.HUS2_AS01_BE01_CF6	INT	0	2359	0	2359	HHMM		Tidkanal BE01 Frånslag 1 Lördag			*)	
		HUS2_AS01_BE01_CF7	AT%MB1148	:INT;	(*	HUS2_AS01_BE01_CF7	AS01	GVL.HUS2_AS01_BE01_CF7	INT	0	2359	0	2359	HHMM		Tidkanal BE01 Frånslag 1 Söndag			*)	
		HUS2_AS01_BE01_CF8	AT%MB1150	:INT;	(*	HUS2_AS01_BE01_CF8	AS01	GVL.HUS2_AS01_BE01_CF8	INT	0	2359	0	2359	HHMM		Tidkanal BE01 Frånslag 1 Helgafton			*)	
		HUS2_AS01_BE01_CF9	AT%MB1152	:INT;	(*	HUS2_AS01_BE01_CF9	AS01	GVL.HUS2_AS01_BE01_CF9	INT	0	2359	0	2359	HHMM		Tidkanal BE01 Frånslag 1 Helgdag			*)	
		HUS2_AS01_BE01_CF11	AT%MB1154	:INT;	(*	HUS2_AS01_BE01_CF11	AS01	GVL.HUS2_AS01_BE01_CF11	INT	0	2359	0	2359	HHMM		Tidkanal BE01 Frånslag 2 Måndag			*)	
		HUS2_AS01_BE01_CF12	AT%MB1156	:INT;	(*	HUS2_AS01_BE01_CF12	AS01	GVL.HUS2_AS01_BE01_CF12	INT	0	2359	0	2359	HHMM		Tidkanal BE01 Frånslag 2 Tisdag			*)	
		HUS2_AS01_BE01_CF13	AT%MB1158	:INT;	(*	HUS2_AS01_BE01_CF13	AS01	GVL.HUS2_AS01_BE01_CF13	INT	0	2359	0	2359	HHMM		Tidkanal BE01 Frånslag 2 Onsdag			*)	
		HUS2_AS01_BE01_CF14	AT%MB1160	:INT;	(*	HUS2_AS01_BE01_CF14	AS01	GVL.HUS2_AS01_BE01_CF14	INT	0	2359	0	2359	HHMM		Tidkanal BE01 Frånslag 2 Torsdag			*)	
		HUS2_AS01_BE01_CF15	AT%MB1162	:INT;	(*	HUS2_AS01_BE01_CF15	AS01	GVL.HUS2_AS01_BE01_CF15	INT	0	2359	0	2359	HHMM		Tidkanal BE01 Frånslag 2 Fredag			*)	
		HUS2_AS01_BE01_CF16	AT%MB1164	:INT;	(*	HUS2_AS01_BE01_CF16	AS01	GVL.HUS2_AS01_BE01_CF16	INT	0	2359	0	2359	HHMM		Tidkanal BE01 Frånslag 2 Lördag			*)	
		HUS2_AS01_BE01_CF17	AT%MB1166	:INT;	(*	HUS2_AS01_BE01_CF17	AS01	GVL.HUS2_AS01_BE01_CF17	INT	0	2359	0	2359	HHMM		Tidkanal BE01 Frånslag 2 Söndag			*)	
		HUS2_AS01_BE01_CF18	AT%MB1168	:INT;	(*	HUS2_AS01_BE01_CF18	AS01	GVL.HUS2_AS01_BE01_CF18	INT	0	2359	0	2359	HHMM		Tidkanal BE01 Frånslag 2 Helgafton			*)	
		HUS2_AS01_BE01_CF19	AT%MB1170	:INT;	(*	HUS2_AS01_BE01_CF19	AS01	GVL.HUS2_AS01_BE01_CF19	INT	0	2359	0	2359	HHMM		Tidkanal BE01 Frånslag 2 Helgdag			*)	
		HUS2_AS01_BE01_MAN	AT%MB1172	:INT;	(*	HUS2_AS01_BE01_MAN	AS01	GVL.HUS2_AS01_BE01_MAN	INT	0	2	0	2			Manuell styrning tidkanal BE01 0=Auto 1=Från 2=Till			*)	
		HUS2_AS01_BE01_FLM	AT%MB1174	:INT;	(*	HUS2_AS01_BE01_FLM	AS01	GVL.HUS2_AS01_BE01_FLM	INT	0	3600	0	3600	Min		Larmfördröjning tidkanal BE01 ej i AUTO			*)	
																				
																				
	(* Tidkanal belysning reserv *)																			
		HUS2_AS01_BE02_CT1	AT%MB1180	:INT;	(*	HUS2_AS01_BE02_CT1	AS01	GVL.HUS2_AS01_BE02_CT1	INT	0	2359	0	2359	HHMM		Tidkanal BE02 Tillslag 1 Måndag			*)	
		HUS2_AS01_BE02_CT2	AT%MB1182	:INT;	(*	HUS2_AS01_BE02_CT2	AS01	GVL.HUS2_AS01_BE02_CT2	INT	0	2359	0	2359	HHMM		Tidkanal BE02 Tillslag 1 Tisdag			*)	
		HUS2_AS01_BE02_CT3	AT%MB1184	:INT;	(*	HUS2_AS01_BE02_CT3	AS01	GVL.HUS2_AS01_BE02_CT3	INT	0	2359	0	2359	HHMM		Tidkanal BE02 Tillslag 1 Onsdag			*)	
		HUS2_AS01_BE02_CT4	AT%MB1186	:INT;	(*	HUS2_AS01_BE02_CT4	AS01	GVL.HUS2_AS01_BE02_CT4	INT	0	2359	0	2359	HHMM		Tidkanal BE02 Tillslag 1 Torsdag			*)	
		HUS2_AS01_BE02_CT5	AT%MB1188	:INT;	(*	HUS2_AS01_BE02_CT5	AS01	GVL.HUS2_AS01_BE02_CT5	INT	0	2359	0	2359	HHMM		Tidkanal BE02 Tillslag 1 Fredag			*)	
		HUS2_AS01_BE02_CT6	AT%MB1190	:INT;	(*	HUS2_AS01_BE02_CT6	AS01	GVL.HUS2_AS01_BE02_CT6	INT	0	2359	0	2359	HHMM		Tidkanal BE02 Tillslag 1 Lördag			*)	
		HUS2_AS01_BE02_CT7	AT%MB1192	:INT;	(*	HUS2_AS01_BE02_CT7	AS01	GVL.HUS2_AS01_BE02_CT7	INT	0	2359	0	2359	HHMM		Tidkanal BE02 Tillslag 1 Söndag			*)	
		HUS2_AS01_BE02_CT8	AT%MB1194	:INT;	(*	HUS2_AS01_BE02_CT8	AS01	GVL.HUS2_AS01_BE02_CT8	INT	0	2359	0	2359	HHMM		Tidkanal BE02 Tillslag 1 Helgafton			*)	
		HUS2_AS01_BE02_CT9	AT%MB1196	:INT;	(*	HUS2_AS01_BE02_CT9	AS01	GVL.HUS2_AS01_BE02_CT9	INT	0	2359	0	2359	HHMM		Tidkanal BE02 Tillslag 1 Helgdag			*)
		HUS2_AS01_BE02_CT11	AT%MB1198	:INT;	(*	HUS2_AS01_BE02_CT11	AS01	GVL.HUS2_AS01_BE02_CT11	INT	0	2359	0	2359	HHMM		Tidkanal BE02 Tillslag 2 Måndag			*)	
		HUS2_AS01_BE02_CT12	AT%MB1200	:INT;	(*	HUS2_AS01_BE02_CT12	AS01	GVL.HUS2_AS01_BE02_CT12	INT	0	2359	0	2359	HHMM		Tidkanal BE02 Tillslag 2 Tisdag			*)	
		HUS2_AS01_BE02_CT13	AT%MB1202	:INT;	(*	HUS2_AS01_BE02_CT13	AS01	GVL.HUS2_AS01_BE02_CT13	INT	0	2359	0	2359	HHMM		Tidkanal BE02 Tillslag 2 Onsdag			*)	
		HUS2_AS01_BE02_CT14	AT%MB1204	:INT;	(*	HUS2_AS01_BE02_CT14	AS01	GVL.HUS2_AS01_BE02_CT14	INT	0	2359	0	2359	HHMM		Tidkanal BE02 Tillslag 2 Torsdag			*)	
		HUS2_AS01_BE02_CT15	AT%MB1206	:INT;	(*	HUS2_AS01_BE02_CT15	AS01	GVL.HUS2_AS01_BE02_CT15	INT	0	2359	0	2359	HHMM		Tidkanal BE02 Tillslag 2 Fredag			*)	
		HUS2_AS01_BE02_CT16	AT%MB1208	:INT;	(*	b	AS01	GVL.HUS2_AS01_BE02_CT16	INT	0	2359	0	2359	HHMM		Tidkanal BE02 Tillslag 2 Lördag			*)	
		HUS2_AS01_BE02_CT17	AT%MB1210	:INT;	(*	HUS2_AS01_BE02_CT17	AS01	GVL.HUS2_AS01_BE02_CT17	INT	0	2359	0	2359	HHMM		Tidkanal BE02 Tillslag 2 Söndag			*)	
		HUS2_AS01_BE02_CT18	AT%MB1212	:INT;	(*	HUS2_AS01_BE02_CT18	AS01	GVL.HUS2_AS01_BE02_CT18	INT	0	2359	0	2359	HHMM		Tidkanal BE02 Tillslag 2 Helgafton			*)	
		HUS2_AS01_BE02_CT19	AT%MB1214	:INT;	(*	HUS2_AS01_BE02_CT19	AS01	GVL.HUS2_AS01_BE02_CT19	INT	0	2359	0	2359	HHMM		Tidkanal BE02 Tillslag 2 Helgdag			*)	
		HUS2_AS01_BE02_CF1	AT%MB1216	:INT;	(*	HUS2_AS01_BE02_CF1	AS01	GVL.HUS2_AS01_BE02_CF1	INT	0	2359	0	2359	HHMM		Tidkanal BE02 Frånslag 1 Måndag			*)	
		HUS2_AS01_BE02_CF2	AT%MB1218	:INT;	(*	HUS2_AS01_BE02_CF2	AS01	GVL.HUS2_AS01_BE02_CF2	INT	0	2359	0	2359	HHMM		Tidkanal BE02 Frånslag 1 Tisdag			*)	
		HUS2_AS01_BE02_CF3	AT%MB1220	:INT;	(*	HUS2_AS01_BE02_CF3	AS01	GVL.HUS2_AS01_BE02_CF3	INT	0	2359	0	2359	HHMM		Tidkanal BE02 Frånslag 1 Onsdag			*)	
		HUS2_AS01_BE02_CF4	AT%MB1222	:INT;	(*	HUS2_AS01_BE02_CF4	AS01	GVL.HUS2_AS01_BE02_CF4	INT	0	2359	0	2359	HHMM		Tidkanal BE02 Frånslag 1 Torsdag			*)	
		HUS2_AS01_BE02_CF5	AT%MB1224	:INT;	(*	HUS2_AS01_BE02_CF5	AS01	GVL.HUS2_AS01_BE02_CF5	INT	0	2359	0	2359	HHMM		Tidkanal BE02 Frånslag 1 Fredag			*)	
		HUS2_AS01_BE02_CF6	AT%MB1226	:INT;	(*	HUS2_AS01_BE02_CF6	AS01	GVL.HUS2_AS01_BE02_CF6	INT	0	2359	0	2359	HHMM		Tidkanal BE02 Frånslag 1 Lördag			*)	
		HUS2_AS01_BE02_CF7	AT%MB1228	:INT;	(*	HUS2_AS01_BE02_CF7	AS01	GVL.HUS2_AS01_BE02_CF7	INT	0	2359	0	2359	HHMM		Tidkanal BE02 Frånslag 1 Söndag			*)	
		HUS2_AS01_BE02_CF8	AT%MB1230	:INT;	(*	HUS2_AS01_BE02_CF8	AS01	GVL.HUS2_AS01_BE02_CF8	INT	0	2359	0	2359	HHMM		Tidkanal BE02 Frånslag 1 Helgafton			*)	
		HUS2_AS01_BE02_CF9	AT%MB1232	:INT;	(*	HUS2_AS01_BE02_CF9	AS01	GVL.HUS2_AS01_BE02_CF9	INT	0	2359	0	2359	HHMM		Tidkanal BE02 Frånslag 1 Helgdag			*)	
		HUS2_AS01_BE02_CF11	AT%MB1234	:INT;	(*	HUS2_AS01_BE02_CF11	AS01	GVL.HUS2_AS01_BE02_CF11	INT	0	2359	0	2359	HHMM		Tidkanal BE02 Frånslag 2 Måndag			*)	
		HUS2_AS01_BE02_CF12	AT%MB1236	:INT;	(*	HUS2_AS01_BE02_CF12	AS01	GVL.HUS2_AS01_BE02_CF12	INT	0	2359	0	2359	HHMM		Tidkanal BE02 Frånslag 2 Tisdag			*)	
		HUS2_AS01_BE02_CF13	AT%MB1238	:INT;	(*	HUS2_AS01_BE02_CF13	AS01	GVL.HUS2_AS01_BE02_CF13	INT	0	2359	0	2359	HHMM		Tidkanal BE02 Frånslag 2 Onsdag			*)	
		HUS2_AS01_BE02_CF14	AT%MB1240	:INT;	(*	HUS2_AS01_BE02_CF14	AS01	GVL.HUS2_AS01_BE02_CF14	INT	0	2359	0	2359	HHMM		Tidkanal BE02 Frånslag 2 Torsdag			*)	
		HUS2_AS01_BE02_CF15	AT%MB1242	:INT;	(*	HUS2_AS01_BE02_CF15	AS01	GVL.HUS2_AS01_BE02_CF15	INT	0	2359	0	2359	HHMM		Tidkanal BE02 Frånslag 2 Fredag			*)	
		HUS2_AS01_BE02_CF16	AT%MB1244	:INT;	(*	HUS2_AS01_BE02_CF16	AS01	GVL.HUS2_AS01_BE02_CF16	INT	0	2359	0	2359	HHMM		Tidkanal BE02 Frånslag 2 Lördag			*)	
		HUS2_AS01_BE02_CF17	AT%MB1246	:INT;	(*	HUS2_AS01_BE02_CF17	AS01	GVL.HUS2_AS01_BE02_CF17	INT	0	2359	0	2359	HHMM		Tidkanal BE02 Frånslag 2 Söndag			*)	
		HUS2_AS01_BE02_CF18	AT%MB1248	:INT;	(*	HUS2_AS01_BE02_CF18	AS01	GVL.HUS2_AS01_BE02_CF18	INT	0	2359	0	2359	HHMM		Tidkanal BE02 Frånslag 2 Helgafton			*)	
		HUS2_AS01_BE02_CF19	AT%MB1250	:INT;	(*	HUS2_AS01_BE02_CF19	AS01	GVL.HUS2_AS01_BE02_CF19	INT	0	2359	0	2359	HHMM		Tidkanal BE02 Frånslag 2 Helgdag			*)	
		HUS2_AS01_BE02_MAN	AT%MB1252	:INT;	(*	HUS2_AS01_BE02_MAN	AS01	GVL.HUS2_AS01_BE02_MAN	INT	0	2	0	2			Manuell styrning tidkanal BE02 0=Auto 1=Från 2=Till			*)	
		HUS2_AS01_BE02_FLM	AT%MB1254	:INT;	(*	HUS2_AS01_BE02_FLM	AS01	GVL.HUS2_AS01_BE02_FLM	INT	0	3600	0	3600	Min		Larmfördröjning tidkanal BE02 ej i AUTO			*)	
																				
																				
		HUS2_AS01_TK01_HHMM	AT%MB1290	:INT;	(*	HUS2_AS01_TK01_HHMM	AS01	GVL.HUS2_AS01_TK01_HHMM	INT	0	2359	0	2359	HHMM		Starttid av motionering AS01 HHMM			*)
		HUS2_AS01_TK01_HHMM1	AT%MB1292	:INT;	(*	HUS2_AS01_TK01_HHMM1	AS01	GVL.HUS2_AS01_TK01_HHMM1	INT	0	2359	0	2359	HHMM		Stopptid av motionering AS01 HHMM			*)
		HUS2_AS01_TK01_VDAG	AT%MB1294	:INT;	(*	HUS2_AS01_TK01_VDAG	AS01	GVL.HUS2_AS01_TK01_VDAG	INT	0	6	0	6	Veckodag		Veckodag för motionering AS01 (0=Sön..6=Lör)			*)	
		HUS2_AS01_TK01_MAN	AT%MB1296	:INT;	(*	HUS2_AS01_TK01_MAN	AS01	GVL.HUS2_AS01_TK01_MAN	INT	0	2	0	2			Manuell styrning motormotionering 0=Auto, 1=Manuell från, 2=Manuell till			*)	
		HUS2_AS01_TK01_FLM	AT%MB1298	:INT;	(*	HUS2_AS01_TK01_FLM	AS01	GVL.HUS2_AS01_TK01_FLM	INT	0	3600	0	3600	Min		Larmfördröjning motormotionering ej i AUTO			*)

		HUS2_AS01_GX31_STAG	AT%MB1300	:REAL;	(*	HUS2_AS01_GX31_STAG	AS01	GVL.HUS2_AS01_GX31_STAG	REAL	0	2000	0	2000	lux		Gränsvärde BE01 belysning TILL			*)
		HUS2_AS01_GX31_STOG	AT%MB1304	:REAL;	(*	HUS2_AS01_GX31_STOG	AS01	GVL.HUS2_AS01_GX31_STOG	REAL	0	2000	0	2000	lux		Gränsvärde BE01 belysning FRÅN			*)	
		HUS2_AS01_GX31_TFD	AT%MB1308	:INT;	(*	HUS2_AS01_GX31_TFD	AS01	GVL.HUS2_AS01_GX31_TFD	INT	0	3600	0	3600	min		Tillslagsfördröjning BE01 belysning TILL			*)	
		HUS2_AS01_GX31_FFD	AT%MB1310	:INT;	(*	HUS2_AS01_GX31_FFD	AS01	GVL.HUS2_AS01_GX31_FFD	INT	0	3600	0	3600	min		Frånslagsfördröjning BE01 belysning FRÅN			*)	
		HUS2_AS01_GX31_STAG1	AT%MB1312	:REAL;	(*	HUS2_AS01_GX31_STAG1	AS01	GVL.HUS2_AS01_GX31_STAG1	REAL	0	2000	0	2000	lux		Gränsvärde BE02 belysning TILL			*)	
		HUS2_AS01_GX31_STOG1	AT%MB1316	:REAL;	(*	HUS2_AS01_GX31_STOG1	AS01	GVL.HUS2_AS01_GX31_STOG1	REAL	0	2000	0	2000	lux		Gränsvärde BE02 belysning FRÅN			*)	
		HUS2_AS01_GX31_TFD1	AT%MB1320	:INT;	(*	HUS2_AS01_GX31_TFD1	AS01	GVL.HUS2_AS01_GX31_TFD1	INT	0	3600	0	3600	min		Tillslagsfördröjning BE02 belysning TILL			*)	
		HUS2_AS01_GX31_FFD1	AT%MB1322	:INT;	(*	HUS2_AS01_GX31_FFD1	AS01	GVL.HUS2_AS01_GX31_FFD1	INT	0	3600	0	3600	min		Frånslagsfördröjning BE02 belysning FRÅN			*)	
																				
																				
		HUS2_AS01_GT31_STAG	AT%MB1324	:REAL;	(*	HUS2_AS01_GT31_STAG	AS01	GVL.HUS2_AS01_GT31_STAG	REAL	0	30	0	30	°C		Gränsvärde pumpstart			*)	
		HUS2_AS01_GT31_STOG	AT%MB1328	:REAL;	(*	HUS2_AS01_GT31_STOG	AS01	GVL.HUS2_AS01_GT31_STOG	REAL	0	30	0	30	°C		Gränsvärde pumpstopp			*)
		HUS2_AS01_GT31_STAG1	AT%MB1332	:REAL;	(*	HUS2_AS01_GT31_STAG1	AS01	GVL.HUS2_AS01_GT31_STAG1	REAL	0	30	0	30	°C		Gränsvärde forcering vintertid			*)
		HUS2_AS01_GT31_STOG1	AT%MB1336	:REAL;	(*	HUS2_AS01_GT31_STOG1	AS01	GVL.HUS2_AS01_GT31_STOG1	REAL	0	30	0	30	°C		Gränsvärde forcering sommartid			*)
		HUS2_AS01_GT3N_TFD	AT%MB1340	:INT;	(*	HUS2_AS01_GT3N_TFD	AS01	GVL.HUS2_AS01_GT3N_TFD	INT	0	3600	0	3600	min		Tillslagsfördröjning pumpstart			*)
		HUS2_AS01_GT3N_FFD	AT%MB1342	:INT;	(*	HUS2_AS01_GT3N_FFD	AS01	GVL.HUS2_AS01_GT3N_FFD	INT	0	3600	0	3600	min		Frånslagsfördröjning pumpstart			*)
		HUS2_AS01_GT3N_FT	AT%MB1344	:INT;	(*	HUS2_AS01_GT3N_FT	AS01	GVL.HUS2_AS01_GT3N_FT	INT	0	3600	0	3600	min		Filtreringstid			*)
																			

		HUS2_AS01_AS02_LC_FL	AT%MB1346	:INT;	(*	HUS2_AS01_AS02_LC_FL	AS01	GVL.HUS2_AS01_AS02_LC_FL	INT	0	3600	0	3600	min		Larmfördröjning kommunikationsfel			*)
		HUS2_AS01_AS03_LC_FL	AT%MB1348	:INT;	(*	HUS2_AS01_AS03_LC_FL	AS01	GVL.HUS2_AS01_AS03_LC_FL	INT	0	3600	0	3600	min		Larmfördröjning kommunikationsfel			*)
		HUS2_AS01_LA01_LC_FL	AT%MB1350	:INT;	(*	HUS2_AS01_LA01_LC_FL	AS01	GVL.HUS2_AS01_LA01_LC_FL	INT	0	3600	0	3600	min		Larmfördröjning kommunikationsfel			*)
		HUS2_AS01_LA02_LC_FL	AT%MB1352	:INT;	(*	HUS2_AS01_LA02_LC_FL	AS01	GVL.HUS2_AS01_LA02_LC_FL	INT	0	3600	0	3600	min		Larmfördröjning kommunikationsfel			*)
		HUS2_AS01_LA03_LC_FL	AT%MB1354	:INT;	(*	HUS2_AS01_LA03_LC_FL	AS01	GVL.HUS2_AS01_LA03_LC_FL	INT	0	3600	0	3600	min		Larmfördröjning kommunikationsfel			*)

		HUS2_AS01_GT31_KRV	AT%MB1356	:INT;	(*	HUS2_AS01_GT31_KRV	AS01	GVL.HUS2_AS01_GT31_KRV	REAL	-10	10	-10	10	°C	0.0	Kalibreringsvärde utetemperatur			*)
		HUS2_AS01_GT3N_GV	AT%MB1360	:REAL;	(*	HUS2_AS01_GT3N_GV	AS01	GVL.HUS2_AS01_GT3N_FT	REAL	0	10	0	10	°C	0.0	Förändring i utetemperatur för uppdatering av GT3N			*)

																				


	END_VAR
																
																

(* Global variable list: HUS2/AS01/HUS2_AS01_IO_Hardvara *)
VAR_GLOBAL


									
	(* Digitala in, KL1488  *)								
	(*Kort1*)								
		AS01_Kort01_DI01				AT %I*			:BOOL;
		AS01_Kort01_DI02				AT %I*			:BOOL;
		AS01_Kort01_DI03				AT %I*			:BOOL;
		AS01_Kort01_DI04				AT %I*			:BOOL;
		AS01_Kort01_DI05				AT %I*			:BOOL;
		AS01_Kort01_DI06				AT %I*			:BOOL;
		AS01_Kort01_DI07				AT %I*			:BOOL;
		AS01_Kort01_DI08				AT %I*			:BOOL;
									
									
	(* Digitala in, KL1488  *)								
	(*Kort2*)								
		AS01_Kort02_DI01				AT %I*			:BOOL;
		AS01_Kort02_DI02				AT %I*			:BOOL;
		AS01_Kort02_DI03				AT %I*			:BOOL;
		AS01_Kort02_DI04				AT %I*			:BOOL;
		AS01_Kort02_DI05				AT %I*			:BOOL;
		AS01_Kort02_DI06				AT %I*			:BOOL;
		AS01_Kort02_DI07				AT %I*			:BOOL;
		AS01_Kort02_DI08				AT %I*			:BOOL;
									
									
	(* Digitala in, KL1488  *)								
	(*Kort3*)								
		AS01_Kort03_DI01				AT %I*			:BOOL;
		AS01_Kort03_DI02				AT %I*			:BOOL;
		AS01_Kort03_DI03				AT %I*			:BOOL;
		AS01_Kort03_DI04				AT %I*			:BOOL;
		AS01_Kort03_DI05				AT %I*			:BOOL;
		AS01_Kort03_DI06				AT %I*			:BOOL;
		AS01_Kort03_DI07				AT %I*			:BOOL;
		AS01_Kort03_DI08				AT %I*			:BOOL;
									
									
	(* Digital Ut, KL2408 *)								
	(*Kort4*)								
		AS01_Kort04_DU01				AT %Q*			:BOOL;
		AS01_Kort04_DU02				AT %Q*			:BOOL;
		AS01_Kort04_DU03				AT %Q*			:BOOL;
		AS01_Kort04_DU04				AT %Q*			:BOOL;
		AS01_Kort04_DU05				AT %Q*			:BOOL;
		AS01_Kort04_DU06				AT %Q*			:BOOL;
		AS01_Kort04_DU07				AT %Q*			:BOOL;
		AS01_Kort04_DU08				AT %Q*			:BOOL;
									
									
	(*Kort5*)								
		AS01_Kort05_DU01				AT %Q*			:BOOL;
		AS01_Kort05_DU02				AT %Q*			:BOOL;
		AS01_Kort05_DU03				AT %Q*			:BOOL;
		AS01_Kort05_DU04				AT %Q*			:BOOL;
		AS01_Kort05_DU05				AT %Q*			:BOOL;
		AS01_Kort05_DU06				AT %Q*			:BOOL;
		AS01_Kort05_DU07				AT %Q*			:BOOL;
		AS01_Kort05_DU08				AT %Q*			:BOOL;
									
									
									
(*	(* Analoga in, KL3208-0010, PT1000 *)								
	(*Kort5*)								
		AS01_Kort06_AI01							
		AS01_Kort06_AI02							
		AS01_Kort06_AI03							
		AS01_Kort06_AI04							
		AS01_Kort06_AI05							
		AS01_Kort06_AI06							
		AS01_Kort06_AI07							
		AS01_Kort06_AI08							
									
									
	(* Analoga in, KL3208-0010, PT1000 *)								
	(*Kort6*)								
		AS01_Kort07_AI01							
		AS01_Kort07_AI02							
		AS01_Kort07_AI03							
		AS01_Kort07_AI04							
		AS01_Kort07_AI05							
		AS01_Kort07_AI06							
		AS01_Kort07_AI07							
		AS01_Kort07_AI08	*)						
									
									
	(* Analoga in, KL3464, 0-10V *)								
	(*Kort7*)								
		AS01_Kort08_AI01				AT %I*			:INT;
		AS01_Kort08_AI02				AT %I*			:INT;
		AS01_Kort08_AI03				AT %I*			:INT;
		AS01_Kort08_AI04				AT %I*			:INT;
									

	(* Analoga ut, KL4408  *)
	(*Kort8*)								
		AS01_Kort09_AU01				AT %Q*			:INT;
		AS01_Kort09_AU02				AT %Q*			:INT;
		AS01_Kort09_AU03				AT %Q*			:INT;
		AS01_Kort09_AU04				AT %Q*			:INT;
		AS01_Kort09_AU05				AT %Q*			:INT;
		AS01_Kort09_AU06				AT %Q*			:INT;
		AS01_Kort09_AU07				AT %Q*			:INT;
		AS01_Kort09_AU08				AT %Q*			:INT;



END_VAR

(* Global variable list: HUS2/AS01/HUS2_AS01_IO_Program *)
VAR_GLOBAL

				(*	Name	Device	Address	Data type	Rawmin	Rawmax	Engmin	Engmax	Unit	Format	Description	Alarmoptions	Trendoptions	*)
	(* Digitala in, KL1488  *)
	(*Kort 1*)
		HUS2_AS01_FB01_L	AT%MX100.0	:BOOL;	(*	HUS2_AS01_FB01_L	AS01	HUS2_AS01_IO_Program.HUS2_AS01_FB01_L	DIGITAL	0	0	0	0			Fasbrott/fel fasföljd	p:A		*)
		HUS2_AS01_JFB01_L	AT%MX100.1	:BOOL;	(*	HUS2_AS01_JFB01_L	AS01	HUS2_AS01_IO_Program.HUS2_AS01_JFB01_L	DIGITAL	0	0	0	0			Jordfelsbrytare 	p:B		*)
		HUS2_AS01_LR01_L	AT%MX100.2	:BOOL;	(*	HUS2_AS01_LR01_L	AS01	HUS2_AS01_IO_Program.HUS2_AS01_LR01_L	DIGITAL	0	0	0	0			Utlöst dvärgbrytare 	p:B		*)
		HUS2_AS01_FS01_L	AT%MX100.3	:BOOL;	(*	HUS2_AS01_FS01_L	AS01	HUS2_AS01_IO_Program.HUS2_AS01_FS01_L	DIGITAL	0	0	0	0			Utlöst finsäkring 	p:B		*)
		HUS2_AS01_RESERV_DI_KORT01_CH05	AT%MX100.4	:BOOL;	(*		AS01									Reserv 			*)
		HUS2_AS01_FP01_L	AT%MX100.5	:BOOL;	(*	HUS2_AS01_FP01_L	AS01	HUS2_AS01_IO_Program.HUS2_AS01_FP01_L	DIGITAL	0	0	0	0			Fellarm strömförsörjn. passersystem	p:B		*)
		HUS2_AS01_VO01_L	AT%MX100.6	:BOOL;	(*	HUS2_AS01_VO01_L	AS01	HUS2_AS01_IO_Program.HUS2_AS01_VO01_L	DIGITAL	0	0	0	0			Utlöst överspänningsskydd	p:B		*)
		HUS2_KV1_PPA201_L	AT%MX100.7	:BOOL;	(*	HUS2_KV1_PPA201_L	AS01	HUS2_AS01_IO_Program.HUS2_KV1_PPA201_L	DIGITAL	0	0	0	0			Summalarm tryckstegringspump	p:B		*)


	(* Digitala in, KL1488  *)
	(*Kort 2*)																		
		HUS2_VS1_GP41_IND	AT%MX101.0	:BOOL;	(*		AS01									Lågt/högt systemtryck 			*)
		HUS2_VS1_PV01_IT	AT%MX101.1	:BOOL;	(*	HUS2_VS1_PV01_IT	AS01	HUS2_AS01_IO_Program.HUS2_VS1_PV01_IT	DIGITAL	0	0	0	0			Driftindikering cirkulationspump			*)
		HUS2_VVC1_PC01_IT	AT%MX101.2	:BOOL;	(*	HUS2_VVC1_PC01_IT	AS01	HUS2_AS01_IO_Program.HUS2_VVC1_PC01_IT	DIGITAL	0	0	0	0			Driftindikering cirkulationspump			*)
		HUS2_VS30_PV01_IT	AT%MX101.3	:BOOL;	(*	HUS2_VS30_PV01_IT	AS01	HUS2_AS01_IO_Program.HUS2_VS30_PV01_IT	DIGITAL	0	0	0	0			Driftindikering cirkulationspump			*)
		HUS2_FA201_FF01_LD	AT%MX101.4	:BOOL;	(*	HUS2_FA201_FF01_LD	AS01	HUS2_AS01_IO_Program.HUS2_FA201_FF01_LD	DIGITAL	0	0	0	0			Driftfel frånluftsfläkt			*)
		HUS2_FA202_FF01_LD	AT%MX101.5	:BOOL;	(*	HUS2_FA202_FF01_LD	AS01	HUS2_AS01_IO_Program.HUS2_FA202_FF01_LD	DIGITAL	0	0	0	0			Driftfel frånluftsfläkt			*)
		HUS2_FA203_FF01_LD	AT%MX101.6	:BOOL;	(*	HUS2_FA203_FF01_LD	AS01	HUS2_AS01_IO_Program.HUS2_FA203_FF01_LD	DIGITAL	0	0	0	0			Driftfel frånluftsfläkt			*)
		HUS2_AS01_RESERV_DI_KORT02_CH08	AT%MX101.7	:BOOL;	(*											Reserv 			*)
																			
																			
	(* Digitala in, KL1488  *)																		
	(*Kort 3*)																		
		HUS2_LB03_HD73_L	AT%MX102.0	:BOOL;	(*	HUS2_LB03_HD73_L	AS01	HUS2_AS01_IO_Program.HUS2_LB03_HD73_L	DIGITAL	0	0	0	0			Utlöst rökdetektor 	p:A		*)
		HUS2_LB03_HD73_L1	AT%MX102.1	:BOOL;	(*	HUS2_LB03_HD73_L1	AS01	HUS2_AS01_IO_Program.HUS2_LB03_HD73_L1	DIGITAL	0	0	0	0			Servicelarm	p:B		*)
		HUS2_LB03_HD73_L2	AT%MX102.2	:BOOL;	(*	HUS2_LB03_HD73_L2	AS01	HUS2_AS01_IO_Program.HUS2_LB03_HD73_L2	DIGITAL	0	0	0	0			Fellarm 	p:B		*)
		HUS2_LB03_BS204_IO	AT%MX102.3	:BOOL;	(*	HUS2_LB03_BS204_IO	AS01	HUS2_AS01_IO_Program.HUS2_LB03_BS204_IO	DIGITAL	0	0	0	0			Indikering öppet 			*)
		HUS2_LB03_BS204_IS	AT%MX102.4	:BOOL;	(*	HUS2_LB03_BS204_IS	AS01	HUS2_AS01_IO_Program.HUS2_LB03_BS204_IS	DIGITAL	0	0	0	0			Indikering stängt 			*)
		HUS2_AS01_RESERV_DI_KORT03_CH06	AT%MX102.5	:BOOL;	(*											Reserv 			*)
		HUS2_AS01_RESERV_DI_KORT03_CH07	AT%MX102.6	:BOOL;	(*											Reserv 			*)
		HUS2_AS01_RESERV_DI_KORT03_CH08	AT%MX102.7	:BOOL;	(*											Reserv 			*)


	(* Digital Ut, KL2408 *)																			
	(*Kort 4*)																			
		HUS2_AS01_SA01_M	AT%MX103.0	:BOOL;	(*											Summalarm AS01 			*)	
		HUS2_AS01_BE01_M	AT%MX103.1	:BOOL;	(*											Tidkanal belysning fasad 			*)
		HUS2_AS01_BE02_M	AT%MX103.2	:BOOL;	(*											Tidkanal belysning reserv			*)	
		HUS2_VS1_PV01_M	AT%MX103.3	:BOOL;	(*											Manöver			*)	
		HUS2_VVC1_PC01_M	AT%MX103.4	:BOOL;	(*											Manöver			*)	
		HUS2_VS30_PV01_M	AT%MX103.5	:BOOL;	(*											Manöver 			*)	
		HUS2_FA201_FF01_M	AT%MX103.6	:BOOL;	(*											Manöver 			*)	
		HUS2_FA202_FF01_M	AT%MX103.7	:BOOL;	(*											Reserv 			*)	
																				
																				
	(* Digital Ut, KL2408 *)																			
	(*Kort 5*)																			
		HUS2_FA203_FF01_M	AT%MX216.0	:BOOL;	(*														*)	
		HUS2_LB03_BS204_M	AT%MX216.1	:BOOL;	(*														*)	
		HUS2_AS01_RESERV_DU_KORT05_CH03	AT%MX216.2	:BOOL;	(*														*)	
		HUS2_AS01_RESERV_DU_KORT05_CH04	AT%MX216.3	:BOOL;	(*														*)	
		HUS2_AS01_RESERV_DU_KORT05_CH05	AT%MX216.4	:BOOL;	(*														*)	
		HUS2_AS01_RESERV_DU_KORT05_CH06	AT%MX216.5	:BOOL;	(*														*)	
		HUS2_AS01_RESERV_DU_KORT05_CH07	AT%MX216.6	:BOOL;	(*														*)	
		HUS2_AS01_RESERV_DU_KORT05_CH08	AT%MX216.7	:BOOL;	(*														*)	


	(* Analoga in, KL3208-0010, PT1000  *)
	(*Kort 6*)																		
		HUS2_AS01_GT31_MV	AT%MB104	:REAL;	(*	HUS2_AS01_GT31_MV	AS01	HUS2_AS01_IO_Program.HUS2_AS01_GT31_MV	REAL	-50	150	-50	150	°C	0.0	Mätvärde utetemperatur			*)
		HUS2_VV1_GT11_MV	AT%MB108	:REAL;	(*	HUS2_VV1_GT11_MV	AS01	HUS2_AS01_IO_Program.HUS2_VV1_GT11_MV	REAL	-50	150	-50	150	°C	0.0	Mätvärde tilloppstemperatur			*)
		HUS2_VS1_GT11_MV	AT%MB112	:REAL;	(*	HUS2_VS1_GT11_MV	AS01	HUS2_AS01_IO_Program.HUS2_VS1_GT11_MV	REAL	-50	150	-50	150	°C	0.0	Mätvärde tilloppstemperatur			*)
		HUS2_VS1_GT41_MV	AT%MB116	:REAL;	(*	HUS2_VS1_GT41_MV	AS01	HUS2_AS01_IO_Program.HUS2_VS1_GT41_MV	REAL	-50	150	-50	150	°C	0.0	Mätvärde returtemperatur			*)
		HUS2_VVC1_GT41_MV	AT%MB120	:REAL;	(*	HUS2_VVC1_GT41_MV	AS01	HUS2_AS01_IO_Program.HUS2_VVC1_GT41_MV	REAL	-50	150	-50	150	°C	0.0	Mätvärde returtemperatur			*)
		HUS2_KV1_GT41_MV	AT%MB124	:REAL;	(*	HUS2_KV1_GT41_MV	AS01	HUS2_AS01_IO_Program.HUS2_KV1_GT41_MV	REAL	-50	150	-50	150	°C	0.0	Mätvärde kallvattentemperatur			*)
		HUS2_VS30_GT11_MV	AT%MB128	:REAL;	(*	HUS2_VS30_GT11_MV	AS01	HUS2_AS01_IO_Program.HUS2_VS30_GT11_MV	REAL	-50	150	-50	150	°C	0.0	Mätvärde tilloppstemperatur			*)
		HUS2_AS01_RESERV_AI_KORT06_CH08	AT%MB132	:REAL;	(*											Reserv			*)
																			
																			
	(* Analoga in, KL3208-0010, PT1000  *)																		
	(*Kort 7*)																		
		HUS2_VS30_GT41_MV	AT%MB136	:REAL;	(*	HUS2_VS30_GT41_MV	AS01	HUS2_AS01_IO_Program.HUS2_VS30_GT41_MV	REAL	-50	150	-50	150	°C	0.0	Mätvärde returtemperatur			*)
		HUS2_FA201_GT51_MV	AT%MB140	:REAL;	(*	HUS2_FA201_GT51_MV	AS01	HUS2_AS01_IO_Program.HUS2_FA201_GT51_MV	REAL	-50	150	-50	150	°C	0.0	Mätvärde frånluftstemperatur			*)
		HUS2_FA202_GT51_MV	AT%MB144	:REAL;	(*	HUS2_FA202_GT51_MV	AS01	HUS2_AS01_IO_Program.HUS2_FA202_GT51_MV	REAL	-50	150	-50	150	°C	0.0	Mätvärde frånluftstemperatur			*)
		HUS2_FA203_GT51_MV	AT%MB148	:REAL;	(*	HUS2_FA203_GT51_MV	AS01	HUS2_AS01_IO_Program.HUS2_FA203_GT51_MV	REAL	-50	150	-50	150	°C	0.0	Mätvärde frånluftstemperatur			*)
		HUS2_AS01_RESERV_AI_KORT07_CH05	AT%MB152	:REAL;	(*											Reserv			*)
		HUS2_AS01_RESERV_AI_KORT07_CH06	AT%MB156	:REAL;	(*											Reserv			*)
		HUS2_AS01_RESERV_AI_KORT07_CH07	AT%MB160	:REAL;	(*											Reserv			*)
		HUS2_AS01_RESERV_AI_KORT07_CH08	AT%MB164	:REAL;	(*											Reserv			*)
																			
																			
	(* Analoga in, KL3464, 0-10V  *)																		
	(*Kort 8*)																		
		HUS2_AS01_GX31_MV	AT%MB168	:REAL;	(*	HUS2_AS01_GX31_MV	AS01	HUS2_AS01_IO_Program.HUS2_AS01_GX31_MV	REAL	0	2000	0	2000	lux	0.0	Uteljusnivå Lux			*)
		HUS2_VS1_GP41_MV	AT%MB172	:REAL;	(*	HUS2_VS1_GP41_MV		HUS2_AS01_IO_Program.HUS2_VS1_GP41_MV	REAL	0	10	0	10	bar	0.0	Mätvärde tryckgivare			*)
		HUS2_AS01_RESERV_AI_KORT08_CH03	AT%MB176	:REAL;	(*											Reserv			*)
		HUS2_AS01_RESERV_AI_KORT08_CH04	AT%MB180	:REAL;	(*											Reserv			*)
																			
																			
	(* Analoga ut, KL4408  *)																		
	(*Kort 9*)																		
		HUS2_VS1_SV11_R	AT%MB184	:REAL;	(*	HUS2_VS1_SV11_R	AS01	HUS2_AS01_IO_Program.HUS2_VS1_SV11_R	REAL	0	100	0	100	%		Styrsignal ventilställdon			*)
		HUS2_VV1_SV11_R	AT%MB188	:REAL;	(*	HUS2_VV1_SV11_R	AS01	HUS2_AS01_IO_Program.HUS2_VV1_SV11_R	REAL	0	100	0	100	%		Styrsignal ventilställdon			*)
		HUS2_VS30_SV21_R	AT%MB192	:REAL;	(*	HUS2_VS30_SV21_R	AS01	HUS2_AS01_IO_Program.HUS2_VS30_SV21_R	REAL	0	100	0	100	%		Styrsignal ventilställdon			*)
		HUS2_FA201_FF01_R	AT%MB196	:REAL;	(*	HUS2_FA201_FF01_R	AS01	HUS2_AS01_IO_Program.HUS2_FA201_FF01_R	REAL	0	100	0	100	%		Styrsignal frånluftsfläkt			*)
		HUS2_FA202_FF01_R	AT%MB200	:REAL;	(*	HUS2_FA202_FF01_R	AS01	HUS2_AS01_IO_Program.HUS2_FA202_FF01_R	REAL	0	100	0	100	%		Styrsignal frånluftsfläkt			*)
		HUS2_FA203_FF01_R	AT%MB204	:REAL;	(*	HUS2_FA203_FF01_R	AS01	HUS2_AS01_IO_Program.HUS2_FA203_FF01_R	REAL	0	100	0	100	%		Styrsignal frånluftsfläkt			*)
		HUS2_AS01_RESERV_AU_KORT09_CH07	AT%MB208	:REAL;	(*											Reserv			*)
		HUS2_AS01_RESERV_AU_KORT09_CH08	AT%MB212	:REAL;	(*											Reserv			*)
																			
																			
																			
																			

																				
																				


END_VAR

(* Global variable list: HUS2/AS01/HUS2_AS01_LARM *)
VAR_GLOBAL

	(* Larm *)																			
		HUS2_AS01_GT31_LG	AT%MX1600.0	:BOOL;	(*	HUS2_AS01_GT31_LG	AS01	GVL.HUS2_AS01_GT31_LG	DIGITAL	0	0	0	0			Givarfel utegivare	p:B		*)
		HUS2_AS01_GX31_LG	AT%MX1600.1	:BOOL;	(*	HUS2_AS01_GX31_LG	AS01	GVL.HUS2_AS01_GX31_LG	DIGITAL	0	0	0	0			Givarfel luxgivare	p:B		*)	
		HUS2_AS01_TK01_LM	AT%MX1600.2	:BOOL;	(*	HUS2_AS01_TK01_LM	AS01	GVL.HUS2_AS01_TK01_LM	DIGITAL	0	0	0	0			Larm pumpmotionering ej i AUTO	p:C		*)
		HUS2_AS01_BE01_LM	AT%MX1600.3	:BOOL;	(*	HUS2_AS01_BE01_LM	AS01	GVL.HUS2_AS01_BE01_LM	DIGITAL	0	0	0	0			Larm tidkanal BE01 ej i AUTO	p:C		*)	
		HUS2_AS01_BE02_LM	AT%MX1600.4	:BOOL;	(*	HUS2_AS01_BE02_LM	AS01	GVL.HUS2_AS01_BE02_LM	DIGITAL	0	0	0	0			Larm tidkanal BE02 ej i AUTO	p:C		*)	
		HUS2_AS01_AS02_LC	AT%MX1600.5	:BOOL;	(*	HUS2_AS01_AS02_LC	AS01	GVL.HUS2_AS01_AS02_LC	DIGITAL	0	0	0	0			Kommunikationsfel	p:B		*)
		HUS2_AS01_AS03_LC	AT%MX1600.6	:BOOL;	(*	HUS2_AS01_AS03_LC	AS01	GVL.HUS2_AS01_AS03_LC	DIGITAL	0	0	0	0			Kommunikationsfel	p:B		*)	
		HUS2_AS01_AL01_LC	AT%MX1600.7	:BOOL;	(*	HUS2_AS01_AL01_LC	AS01	GVL.HUS2_AS01_AL01_LC	DIGITAL	0	0	0	0			Kommunikationsfel	p:B		*)
		HUS2_AS01_AL02_LC	AT%MX1601.0	:BOOL;	(*	HUS2_AS01_AL02_LC	AS01	GVL.HUS2_AS01_AL02_LC	DIGITAL	0	0	0	0			Kommunikationsfel	p:B		*)	
		HUS2_AS01_AL03_LC	AT%MX1601.1	:BOOL;	(*	HUS2_AS01_AL03_LC	AS01	GVL.HUS2_AS01_AL03_LC	DIGITAL	0	0	0	0			Kommunikationsfel	p:B		*)	
		HUS2_AS01_PLC_L	AT%MX1601.2	:BOOL;	(*	HUS2_AS01_PLC_L	AS01	GVL.HUS2_AS01_PLC_L	DIGITAL	0	0	0	0			IO-fel	p:B		*)	
		HUS2_AS01_PLC_L1	AT%MX1601.3	:BOOL;	(*	HUS2_AS01_PLC_L1	AS01	GVL.HUS2_AS01_PLC_L1	DIGITAL	0	0	0	0			Internt fel	p:B		*)
		HUS2_AS01_PLC_L2	AT%MX1601.4	:BOOL;	(*	HUS2_AS01_PLC_L2	AS01	GVL.HUS2_AS01_PLC_L2	DIGITAL	0	0	0	0			Byt batteri	p:B		*)	
		HUS2_AS01_AS02_L	AT%MX1601.5	:BOOL;	(*	HUS2_AS01_AS02_L	AS01	GVL.HUS2_AS01_AS02_L	DIGITAL	0	0	0	0			IO-fel	p:B		*)
		HUS2_AS01_AS03_L	AT%MX1601.6	:BOOL;	(*	HUS2_AS01_AS03_L	AS01	GVL.HUS2_AS01_AS03_L	DIGITAL	0	0	0	0			IO-fel	p:B		*)
		HUS2_AS01_AL01_L	AT%MX1601.7	:BOOL;	(*	HUS2_AS01_AL01_L	AS01	GVL.HUS2_AS01_AL01_L	DIGITAL	0	0	0	0			IO-fel	p:B		*)
		HUS2_AS01_AL02_L	AT%MX1602.0	:BOOL;	(*	HUS2_AS01_AL02_L	AS01	GVL.HUS2_AS01_AL02_L	DIGITAL	0	0	0	0			IO-fel	p:B		*)
		HUS2_AS01_AL03_L	AT%MX1602.1	:BOOL;	(*	HUS2_AS01_AL03_L	AS01	GVL.HUS2_AS01_AL03_L	DIGITAL	0	0	0	0			IO-fel	p:B		*)
		HUS2_AS01_WEBPORT_M	AT%MX1602.2	:BOOL;	(*Larm	DIGITAL	0	0	0	0			Larm 	p:A		*)
		HUS2_AS01_TEST	AT%MX1602.3	:BOOL;	(*Larm	DIGITAL	0	0	0	0			Larm 	p:A		*)


																				
	(* ACK larm *)
																				
		HUS2_AS01_PLC_L2_ACK	AT%MX1610.0	:BOOL;	(*	HUS2_AS01_PLC_L2_ACK	AS01	GVL.HUS2_AS01_PLC_L2_ACK	DIGITAL	0	0	0	0			Kvittering batterilarm			*)	
																				
																				
																				



END_VAR

(* Global variable list: HUS2/AS01/HUS2_AS01_OVRIGT *)
VAR_GLOBAL


		HUS2_AS01_TK01_IT	AT%MX1620.0	:BOOL;	(*	HUS2_AS01_TK01_IT	AS01	GVL.HUS2_AS01_TK01_IT	DIGITAL	0	0	0	0			Tidkanal TK01 Aktiv			*)
		HUS2_AS01_BE01_IT	AT%MX1620.1	:BOOL;	(*	HUS2_AS01_BE01_IT	AS01	GVL.HUS2_AS01_BE01_IT	DIGITAL	0	0	0	0			Tidkanal BE01 Aktiv 			*)
		HUS2_AS01_BE02_IT	AT%MX1620.2	:BOOL;	(*	HUS2_AS01_BE02_IT	AS01	GVL.HUS2_AS01_BE02_IT	DIGITAL	0	0	0	0			Tidkanal BE02 Aktiv			*)		
		HUS2_AS01_PLCTID_TRIGG	AT%MX1620.3	:BOOL;	(*	HUS2_AS01_PLCTID_TRIGG	AS10	GVL.HUS2_AS01_PLCTID_TRIGG	DIGITAL	0	0	0	0			Puls för skrivning av tid till PLC, Nollställs automatiskt efter skrivning			*)		
																					
																					

																					
																					
																					
																					
																					
	(* Tidshantering i PLC *)																				
		HUS2_AS01_PLCTID_SEK	AT%MB1630	:INT;	(*	HUS2_AS01_PLCTID_SEK	AS01	GVL.HUS2_AS01_PLCTID_SEK	INT	0	60	0	60	Sek		Tid i PLC, Aktuell sekund			*)		
		HUS2_AS01_PLCTID_HHMM	AT%MB1632	:INT;	(*	HUS2_AS01_PLCTID_HHMM	AS01	GVL.HUS2_AS01_PLCTID_HHMM	INT	0	2359	0	2359	HHMM		Tid i PLC, Aktuell minut & timme			*)		
		HUS2_AS01_PLCTID_MMDD	AT%MB1634	:INT;	(*	HUS2_AS01_PLCTID_MMDD	AS01	GVL.HUS2_AS01_PLCTID_MMDD	INT	0	1231	0	1231	MMDD		Tid i PLC, Aktuell månad & dag			*)		
		HUS2_AS01_PLCTID_VDAG	AT%MB1636	:INT;	(*	HUS2_AS01_PLCTID_VDAG	AS01	GVL.HUS2_AS01_PLCTID_VDAG	INT	0	6	0	6	Veckodag		Tid i PLC, Aktuell veckodag			*)		
		HUS2_AS01_PLCTID_YYYY	AT%MB1638	:INT;	(*	HUS2_AS01_PLCTID_YYYY	AS01	GVL.HUS2_AS01_PLCTID_YYYY	INT	0	2359	0	2359	HHMM		Tid i PLC, Aktuell år			*)		
		HUS2_AS01_PLCTID_WSEK	AT%MB1640	:INT;	(*	HUS2_AS01_PLCTID_WSEK	AS01	GVL.HUS2_AS01_PLCTID_WSEK	INT							Tid i PLC, Skriv sekund			*)		
		HUS2_AS01_PLCTID_WMIN	AT%MB1642	:INT;	(*	HUS2_AS01_PLCTID_WMIN	AS01	GVL.HUS2_AS01_PLCTID_WMIN	INT							Tid i PLC, Skriv minut			*)		
		HUS2_AS01_PLCTID_WTIM	AT%MB1644	:INT;	(*	HUS2_AS01_PLCTID_WTIM	AS01	GVL.HUS2_AS01_PLCTID_WTIM	INT							Tid i PLC, Skriv timme			*)		
		HUS2_AS01_PLCTID_WDAG	AT%MB1646	:INT;	(*	HUS2_AS01_PLCTID_WDAG	AS01	GVL.HUS2_AS01_PLCTID_WDAG	INT							Tid i PLC, Skriv datum			*)		
		HUS2_AS01_PLCTID_WMND	AT%MB1648	:INT;	(*	HUS2_AS01_PLCTID_WMND	AS01	GVL.HUS2_AS01_PLCTID_WMND	INT							Tid i PLC, Skriv månad			*)		
		HUS2_AS01_PLCTID_WAR	AT%MB1650	:INT;	(*	HUS2_AS01_PLCTID_WAR	AS01	GVL.HUS2_AS01_PLCTID_WAR	INT							Tid i PLC, Skriv år			*)		

		HUS2_AS01_GT3N_MV	AT%MB1652	:REAL;	(*	HUS2_AS01_GT3N_MV	AS01	GVL.HUS2_AS01_GT3N_MV	REAL	-50	150	-50	150	°C	0.0	Filtrerad utetemperatur			*)

																				

																					

																					

END_VAR

(* Global variable list: HUS2/BS201, BS202, BS203, BS204/HUS2_BS201_204_INST *)
VAR_GLOBAL PERSISTENT



				(*	Name	Device	Address	Data type	Rawmin	Rawmax	Engmin	Engmax	Unit	Format	Description	Alarmoptions	Trendoptions	*)
																			
	HUS2_AS01_BS_HHMM	AT%MB3460	:INT;	(*	HUS2_AS01_BS_HHMM	AS01	GVL.HUS2_AS01_BS_HHMM	INT	0	2359	0	2359	HHMM		Starttid av motionering brandspjäll HHMM			*)
	HUS2_AS01_BS_VDAG	AT%MB3462	:INT;	(*	HUS2_AS01_BS_VDAG	AS01	GVL.HUS2_AS01_BS_VDAG	INT	0	6	0	6	Veckodag		Veckodag för motionering brandspjäll (0=Sön..6=Lör)			*)	
	HUS2_AS01_BS_MAN	AT%MB3464	:INT;	(*	HUS2_AS01_BS_MAN	AS01	GVL.HUS2_AS01_BS_MAN	INT	0	2	0	2			Manuell styrning motionering brandspjäll 0=Auto, 1=Manuell från, 2=Manuell till			*)	
	HUS2_AS01_BS_FLM	AT%MB3466	:INT;	(*	HUS2_AS01_BS_FLM	AS01	GVL.HUS2_AS01_BS_FLM	INT	0	3600	0	3600	Min		Larmfördröjning motionering brandspjäll ej i AUTO			*)	
	HUS2_LB03_BS201_MAN	AT%MB3468	:INT;	(*	HUS2_LB03_BS201_MAN	AS01	GVL.HUS2_LB03_BS201_MAN	INT	0	2	0	2			Manuell styrning brandspjäll 0=Auto,1=Från,2=Till			*)	
	HUS2_LB03_BS201_FLM	AT%MB3470	:INT;	(*	HUS2_LB03_BS201_FLM	AS01	GVL.HUS2_LB03_BS201_FLM	INT	0	3600	0	3600	Min		Larmfördröjning brandspjäll ej i AUTO			*)	
	HUS2_LB03_BS201_FL	AT%MB3472	:INT;	(*	HUS2_LB03_BS201_FL	AS01	GVL.HUS2_LB03_BS201_FL	INT	0	1000	0	1000	Sek		Larmfördröjning brandspjäll öppnar ej			*)	
	HUS2_LB03_BS201_FL1	AT%MB3474	:INT;	(*	HUS2_LB03_BS201_FL1	AS01	GVL.HUS2_LB03_BS201_FL1	INT	0	1000	0	1000	Sek		Larmfördröjning brandspjäll stänger ej			*)	
	HUS2_LB03_BS202_MAN	AT%MB3476	:INT;	(*	HUS2_LB03_BS202_MAN	AS01	GVL.HUS2_LB03_BS202_MAN	INT	0	2	0	2			Manuell styrning brandspjäll 0=Auto,1=Från,2=Till			*)	
	HUS2_LB03_BS202_FLM	AT%MB3478	:INT;	(*	HUS2_LB03_BS202_FLM	AS01	GVL.HUS2_LB03_BS202_FLM	INT	0	3600	0	3600	Min		Larmfördröjning brandspjäll ej i AUTO			*)	
	HUS2_LB03_BS202_FL	AT%MB3480	:INT;	(*	HUS2_LB03_BS202_FL	AS01	GVL.HUS2_LB03_BS202_FL	INT	0	1000	0	1000	Sek		Larmfördröjning brandspjäll öppnar ej			*)	
	HUS2_LB03_BS202_FL1	AT%MB3482	:INT;	(*	HUS2_LB03_BS202_FL1	AS01	GVL.HUS2_LB03_BS202_FL1	INT	0	1000	0	1000	Sek		Larmfördröjning brandspjäll stänger ej			*)	
	HUS2_LB03_BS203_MAN	AT%MB3484	:INT;	(*	HUS2_LB03_BS203_MAN	AS01	GVL.HUS2_LB03_BS203_MAN	INT	0	2	0	2			Manuell styrning brandspjäll 0=Auto,1=Från,2=Till			*)
	HUS2_LB03_BS203_FLM	AT%MB3486	:INT;	(*	HUS2_LB03_BS203_FLM	AS01	GVL.HUS2_LB03_BS203_FLM	INT	0	3600	0	3600	Min		Larmfördröjning brandspjäll ej i AUTO			*)	
	HUS2_LB03_BS203_FL	AT%MB3488	:INT;	(*	HUS2_LB03_BS203_FL	AS01	GVL.HUS2_LB03_BS203_FL	INT	0	1000	0	1000	Sek		Larmfördröjning brandspjäll öppnar ej			*)	
	HUS2_LB03_BS203_FL1	AT%MB3490	:INT;	(*	HUS2_LB03_BS203_FL1	AS01	GVL.HUS2_LB03_BS203_FL1	INT	0	1000	0	1000	Sek		Larmfördröjning brandspjäll stänger ej			*)	
	HUS2_LB03_BS204_MAN	AT%MB3492	:INT;	(*	HUS2_LB03_BS204_MAN	AS01	GVL.HUS2_LB03_BS204_MAN	INT	0	2	0	2			Manuell styrning brandspjäll 0=Auto,1=Från,2=Till			*)	
	HUS2_LB03_BS204_FLM	AT%MB3494	:INT;	(*	HUS2_LB03_BS204_FLM	AS01	GVL.HUS2_LB03_BS204_FLM	INT	0	3600	0	3600	Min		Larmfördröjning brandspjäll ej i AUTO			*)	
	HUS2_LB03_BS204_FL	AT%MB3496	:INT;	(*	HUS2_LB03_BS204_FL	AS01	GVL.HUS2_LB03_BS204_FL	INT	0	1000	0	1000	Sek		Larmfördröjning brandspjäll öppnar ej			*)	
	HUS2_LB03_BS204_FL1	AT%MB3498	:INT;	(*	HUS2_LB03_BS204_FL1	AS01	GVL.HUS2_LB03_BS204_FL1	INT	0	1000	0	1000	Sek		Larmfördröjning brandspjäll stänger ej			*)	
																			
																			
																			


END_VAR
																
																

(* Global variable list: HUS2/BS201, BS202, BS203, BS204/HUS2_BS201_204_LARM *)
VAR_GLOBAL


																						
	HUS2_AS01_BS_LM	AT%MX3530.0	:BOOL;	(*	HUS2_AS01_BS_LM	AS01	GVL.HUS2_AS01_BS_LM	DIGITAL	0	0	0	0			Larm motionering brandspjäll ej i AUTO	p:C		*)				
	HUS2_LB03_BS201_LM	AT%MX3530.1	:BOOL; 	(*	HUS2_LB03_BS201_LM	AS01	GVL.HUS2_LB03_BS201_LM	DIGITAL	0	0	0	0			Brandspjäll ej i läge AUTO	p:C		*)				
	HUS2_LB03_BS201_L	AT%MX3530.2	:BOOL; 	(*	HUS2_LB03_BS201_L	AS01	GVL.HUS2_LB03_BS201_L	DIGITAL	0	0	0	0			Brandspjäll öppnar ej	p:B		*)
	HUS2_LB03_BS201_L1	AT%MX3530.3	:BOOL; 	(*	HUS2_LB03_BS201_L1	AS01	GVL.HUS2_LB03_BS201_L1	DIGITAL	0	0	0	0			Brandspjäll stänger ej	p:B		*)				
	HUS2_LB03_BS201_L2	AT%MX3530.4	:BOOL; 	(*	HUS2_LB03_BS201_L2	AS01	GVL.HUS2_LB03_BS201_L2	DIGITAL	0	0	0	0			Brandspjäll stängt och öppet samtidigt	p:B		*)				
	HUS2_LB03_BS201_ACK	AT%MX3530.5	:BOOL; 	(*	HUS2_LB03_BS201_ACK	AS01	GVL.HUS2_LB03_BS201_ACK	DIGITAL	0	0	0	0			Larmkvittens brandspjäll BS201			*)				
	HUS2_LB03_BS202_LM	AT%MX3530.6	:BOOL; 	(*	HUS2_LB03_BS202_LM	AS01	GVL.HUS2_LB03_BS202_LM	DIGITAL	0	0	0	0			Brandspjäll ej i läge AUTO	p:C		*)				
	HUS2_LB03_BS202_L	AT%MX3530.7	:BOOL; 	(*	HUS2_LB03_BS202_L	AS01	GVL.HUS2_LB03_BS202_L	DIGITAL	0	0	0	0			Brandspjäll öppnar ej	p:B		*)				
	HUS2_LB03_BS202_L1	AT%MX3531.0	:BOOL; 	(*	HUS2_LB03_BS202_L1	AS01	GVL.HUS2_LB03_BS202_L1	DIGITAL	0	0	0	0			Brandspjäll stänger ej	p:B		*)				
	HUS2_LB03_BS202_L2	AT%MX3531.1	:BOOL; 	(*	HUS2_LB03_BS202_L2	AS01	GVL.HUS2_LB03_BS202_L2	DIGITAL	0	0	0	0			Brandspjäll stängt och öppet samtidigt	p:B		*)				
	HUS2_LB03_BS202_ACK	AT%MX3531.2	:BOOL; 	(*	HUS2_LB03_BS202_ACK	AS01	GVL.HUS2_LB03_BS202_ACK	DIGITAL	0	0	0	0			Larmkvittens brandspjäll BS202			*)				
	HUS2_LB03_BS203_LM	AT%MX3531.3	:BOOL; 	(*	HUS2_LB03_BS203_LM	AS01	GVL.HUS2_LB03_BS203_LM	DIGITAL	0	0	0	0			Brandspjäll ej i läge AUTO	p:C		*)				
	HUS2_LB03_BS203_L	AT%MX3531.4	:BOOL; 	(*	HUS2_LB03_BS203_L	AS01	GVL.HUS2_LB03_BS203_L	DIGITAL	0	0	0	0			Brandspjäll öppnar ej	p:B		*)				
	HUS2_LB03_BS203_L1	AT%MX3531.5	:BOOL; 	(*	HUS2_LB03_BS203_L1	AS01	GVL.HUS2_LB03_BS203_L1	DIGITAL	0	0	0	0			Brandspjäll stänger ej	p:B		*)				
	HUS2_LB03_BS203_L2	AT%MX3531.6	:BOOL; 	(*	HUS2_LB03_BS203_L2	AS01	GVL.HUS2_LB03_BS203_L2	DIGITAL	0	0	0	0			Brandspjäll stängt och öppet samtidigt	p:B		*)				
	HUS2_LB03_BS203_ACK	AT%MX3531.7	:BOOL; 	(*	HUS2_LB03_BS203_ACK	AS01	GVL.HUS2_LB03_BS203_ACK	DIGITAL	0	0	0	0			Larmkvittens brandspjäll BS203			*)				
	HUS2_LB03_BS204_LM	AT%MX3532.0	:BOOL; 	(*	HUS2_LB03_BS204_LM	AS01	GVL.HUS2_LB03_BS204_LM	DIGITAL	0	0	0	0			Brandspjäll ej i läge AUTO	p:C		*)				
	HUS2_LB03_BS204_L	AT%MX3532.1	:BOOL; 	(*	HUS2_LB03_BS204_L	AS01	GVL.HUS2_LB03_BS204_L	DIGITAL	0	0	0	0			Brandspjäll öppnar ej	p:B		*)				
	HUS2_LB03_BS204_L1	AT%MX3532.2	:BOOL; 	(*	HUS2_LB03_BS204_L1	AS01	GVL.HUS2_LB03_BS204_L1	DIGITAL	0	0	0	0			Brandspjäll stänger ej	p:B		*)				
	HUS2_LB03_BS204_L2	AT%MX3532.3	:BOOL; 	(*	HUS2_LB03_BS204_L2	AS01	GVL.HUS2_LB03_BS204_L2	DIGITAL	0	0	0	0			Brandspjäll stängt och öppet samtidigt	p:B		*)				
	HUS2_LB03_BS204_ACK	AT%MX3532.4	:BOOL; 	(*	HUS2_LB03_BS204_ACK	AS01	GVL.HUS2_LB03_BS204_ACK	DIGITAL	0	0	0	0			Larmkvittens brandspjäll BS204			*)				
																						
																						

END_VAR

(* Global variable list: HUS2/BS201, BS202, BS203, BS204/HUS2_BS201_204_OVRIGT *)
VAR_GLOBAL

	HUS2_AS01_BS_IT	AT%MX3536.0	:BOOL;	(*	HUS2_AS01_TK01_IT	AS01	GVL.HUS2_AS01_TK01_IT	DIGITAL	0	0	0	0			Tidkanal motionering brandspjäll Aktiv			*)
	HUS2_LB03_BS201_IT	AT%MX3536.1	:BOOL;	(*	HUS2_LB03_BS201_IT	AS01	GVL.HUS2_LB03_BS201_IT	DIGITAL	0	0	0	0			Motionering aktiv			*)
	HUS2_LB03_BS202_IT	AT%MX3536.2	:BOOL;	(*	HUS2_LB03_BS202_IT	AS01	GVL.HUS2_LB03_BS202_IT	DIGITAL	0	0	0	0			Motionering aktiv			*)
	HUS2_LB03_BS203_IT	AT%MX3536.3	:BOOL;	(*	HUS2_LB03_BS203_IT	AS01	GVL.HUS2_LB03_BS203_IT	DIGITAL	0	0	0	0			Motionering aktiv			*)
	HUS2_LB03_BS204_IT	AT%MX3536.4	:BOOL;	(*	HUS2_LB03_BS204_IT	AS01	GVL.HUS2_LB03_BS204_IT	DIGITAL	0	0	0	0			Motionering aktiv			*)
																									
																									

END_VAR

(* Global variable list: HUS2/FA201, FA202, FA203/HUS2_FA201_203_INST *)
VAR_GLOBAL PERSISTENT


					(*	Name	Device	Address	Data type	Rawmin	Rawmax	Engmin	Engmax	Unit	Format	Description	Alarmoptions	Trendoptions	*)
																			
		HUS2_FA201_SO1_MAN	AT%MB3000	:INT;	(*	HUS2_FA201_SO1_MAN	AS01	GVL.HUS2_FA201_SO1_MAN	INT	0	2	0	2			Manuell styrning system FA201. 0=Auto, 1=Manuell från, 2=Manuell till			*)
		HUS2_FA201_SO1_FLM	AT%MB3002	:INT;	(*	HUS2_FA201_SO1_FLM	AS01	GVL.HUS2_FA201_SO1_FLM	INT	0	3600	0	3600	Min		Larmfördröjning serviceomkopplare ej i läge AUTO			*)
																			
		HUS2_FA201_FF01_FLM	AT%MB3004	:INT;	(*	HUS2_FA201_FF01_FLM	AS01	GVL.HUS2_FA201_FF01_FLM	INT	0	3600	0	3600	Min		Larmfördröjning frånluftsfläkt ej i AUTO			*)
		HUS2_FA201_FF01_FLD	AT%MB3006	:INT;	(*	HUS2_FA201_FF01_FLD	AS01	GVL.HUS2_FA201_FF01_FLD	INT	0	120	0	120	Sek		Larmfördröjning driftfel frånluftsfläkt			*)
																			
		HUS2_FA201_FF01_MAN	AT%MB3008	:INT;	(*	HUS2_FA201_FF01_MAN	AS01	GVL.HUS2_FA201_FF01_MAN	INT	0	2	0	2			Manuell styrning frånluftsfläkt 0=Auto,1=Från,2=Till			*)
		HUS2_FA201_FF01_MAN1	AT%MB3010	:INT;	(*	HUS2_FA201_FF01_MAN	AS01	GVL.HUS2_FA201_FF01_MAN	INT	0	1	0	1			Manuell styrning styrsignal frånluftsfläkt 0=Auto,1=Till			*)
		HUS2_FA201_FF01_RMAN	AT%MB3012	:REAL;	(*	HUS2_FA201_FF01_RMAN	AS01	GVL.HUS2_FA201_FF01_RMAN	REAL	0	100	0	100	%		Manuell styrsignal frånluftsfläkt			*)
																			
		HUS2_FA201_GT51_STAG	AT%MB3016	:REAL;	(*	HUS2_FA201_GT51_STAG	AS01	GVL.HUS2_FA201_GT51_STAG	REAL	0	50	0	50	°C	0.0	Gränsvärde start forcering frånluftsfläkt			*)
		HUS2_FA201_GT51_STOG	AT%MB3020	:REAL;	(*	HUS2_FA201_GT51_STOG	AS01	GVL.HUS2_FA201_GT51_STOG	REAL	0	50	0	50	°C	0.0	Gränsvärde stopp forcering frånluftsfläkt			*)
																			
		HUS2_FA201_GT51_GVH	AT%MB3024	:REAL;	(*	HUS2_FA201_GT51_GVH	AS01	GVL.HUS2_FA201_GT51_GVH	REAL	0	50	0	50	°C	0.0	Gränsvärde hög temperatur			*)
		HUS2_FA201_GT51_FLG	AT%MB3028	:INT;	(*	HUS2_FA201_GT51_FLG	AS01	GVL.HUS2_FA201_GT51_FLG	INT	0	3600	0	3600	Min		Lamfördröjning hög temperatur			*)
																			

		HUS2_FA201_GT51_KRV	AT%MB3036	:REAL;	(*	HUS2_FA201_GT51_KRV	AS01	GVL.HUS2_FA201_GT51_KRV	REAL	-10	10	-10	10	°C	0.0	Kalibreringsvärde frånluftsgivare			*)

		HUS2_FA201_FF01_BV	AT%MB3040	:REAL;	(*	HUS2_FA201_FF01_BV	AS01	GVL.HUS2_FA201_FF01_BV	REAL	0	100	0	100	%		Grundflöde frånluftsfläkt			*)
		HUS2_FA201_FF01_BV1	AT%MB3044	:REAL;	(*	HUS2_FA201_FF01_BV1	AS01	GVL.HUS2_FA201_FF01_BV1	REAL	0	100	0	100	%		Forcerat flöde frånluftsfläkt			*)
																			
																			
																			
																			
																			
																			
		HUS2_FA202_SO1_MAN	AT%MB3060	:INT;	(*	HUS2_FA202_SO1_MAN	AS01	GVL.HUS2_FA202_SO1_MAN	INT	0	2	0	2			Manuell styrning system FA202. 0=Auto, 1=Manuell från, 2=Manuell till			*)
		HUS2_FA202_SO1_FLM	AT%MB3062	:INT;	(*	HUS2_FA202_SO1_FLM	AS01	GVL.HUS2_FA202_SO1_FLM	INT	0	3600	0	3600	Min		Larmfördröjning serviceomkopplare ej i läge AUTO			*)
																			
		HUS2_FA202_FF01_FLM	AT%MB3064	:INT;	(*	HUS2_FA202_FF01_FLM	AS01	GVL.HUS2_FA202_FF01_FLM	INT	0	3600	0	3600	Min		Larmfördröjning frånluftsfläkt ej i AUTO			*)
		HUS2_FA202_FF01_FLD	AT%MB3066	:INT;	(*	HUS2_FA202_FF01_FLD	AS01	GVL.HUS2_FA202_FF01_FLD	INT	0	120	0	120	Sek		Larmfördröjning driftfel frånluftsfläkt			*)
																			
		HUS2_FA202_FF01_MAN	AT%MB3068	:INT;	(*	HUS2_FA202_FF01_MAN	AS01	GVL.HUS2_FA202_FF01_MAN	INT	0	2	0	2			Manuell styrning frånluftsfläkt 0=Auto,1=Från,2=Till			*)
		HUS2_FA202_FF01_MAN1	AT%MB3070	:INT;	(*	HUS2_FA202_FF01_MAN	AS01	GVL.HUS2_FA202_FF01_MAN	INT	0	1	0	1			Manuell styrning styrsignal frånluftsfläkt 0=Auto,1=Till			*)
		HUS2_FA202_FF01_RMAN	AT%MB3072	:REAL;	(*	HUS2_FA202_FF01_RMAN	AS01	GVL.HUS2_FA202_FF01_RMAN	REAL	0	100	0	100	%		Manuell styrsignal frånluftsfläkt			*)
																			
		HUS2_FA202_GT51_STAG	AT%MB3076	:REAL;	(*	HUS2_FA202_GT51_STAG	AS01	GVL.HUS2_FA202_GT51_STAG	REAL	0	50	0	50	°C	0.0	Gränsvärde start forcering frånluftsfläkt			*)
		HUS2_FA202_GT51_STOG	AT%MB3080	:REAL;	(*	HUS2_FA202_GT51_STOG	AS01	GVL.HUS2_FA202_GT51_STOG	REAL	0	50	0	50	°C	0.0	Gränsvärde stopp forcering frånluftsfläkt			*)
																			
		HUS2_FA202_GT51_GVH	AT%MB3084	:REAL;	(*	HUS2_FA202_GT51_GVH	AS01	GVL.HUS2_FA202_GT51_GVH	REAL	0	50	0	50	°C	0.0	Gränsvärde hög temperatur			*)
		HUS2_FA202_GT51_FLG	AT%MB3088	:INT;	(*	HUS2_FA202_GT51_FLG	AS01	GVL.HUS2_FA202_GT51_FLG	INT	0	3600	0	3600	Min		Lamfördröjning hög temperatur			*)
																			

		HUS2_FA202_GT51_KRV	AT%MB3096	:REAL;	(*	HUS2_FA202_GT51_KRV	AS01	GVL.HUS2_FA202_GT51_KRV	REAL	-10	10	-10	10	°C	0.0	Kalibreringsvärde frånluftsgivare			*)
																			
		HUS2_FA202_FF01_BV	AT%MB3100	:REAL;	(*	HUS2_FA202_FF01_BV	AS01	GVL.HUS2_FA202_FF01_BV	REAL	0	100	0	100	%		Grundflöde frånluftsfläkt			*)
		HUS2_FA202_FF01_BV1	AT%MB3104	:REAL;	(*	HUS2_FA202_FF01_BV1	AS01	GVL.HUS2_FA202_FF01_BV1	REAL	0	100	0	100	%		Forcerat flöde frånluftsfläkt			*)
																			
																			
																			
																			
																			
																			
		HUS2_FA203_SO1_MAN	AT%MB3120	:INT;	(*	HUS2_FA203_SO1_MAN	AS01	GVL.HUS2_FA203_SO1_MAN	INT	0	2	0	2			Manuell styrning system FA203. 0=Auto, 1=Manuell från, 2=Manuell till			*)
		HUS2_FA203_SO1_FLM	AT%MB3122	:INT;	(*	HUS2_FA203_SO1_FLM	AS01	GVL.HUS2_FA203_SO1_FLM	INT	0	3600	0	3600	Min		Larmfördröjning serviceomkopplare ej i läge AUTO			*)
																			
		HUS2_FA203_FF01_FLM	AT%MB3124	:INT;	(*	HUS2_FA203_FF01_FLM	AS01	GVL.HUS2_FA203_FF01_FLM	INT	0	3600	0	3600	Min		Larmfördröjning frånluftsfläkt ej i AUTO			*)
		HUS2_FA203_FF01_FLD	AT%MB3126	:INT;	(*	HUS2_FA203_FF01_FLD	AS01	GVL.HUS2_FA203_FF01_FLD	INT	0	120	0	120	Sek		Larmfördröjning driftfel frånluftsfläkt			*)
																			
		HUS2_FA203_FF01_MAN	AT%MB3128	:INT;	(*	HUS2_FA203_FF01_MAN	AS01	GVL.HUS2_FA203_FF01_MAN	INT	0	2	0	2			Manuell styrning frånluftsfläkt 0=Auto,1=Från,2=Till			*)
		HUS2_FA203_FF01_MAN1	AT%MB3130	:INT;	(*	HUS2_FA203_FF01_MAN	AS01	GVL.HUS2_FA203_FF01_MAN	INT	0	1	0	1			Manuell styrning styrsignal frånluftsfläkt 0=Auto,1=Till			*)
		HUS2_FA203_FF01_RMAN	AT%MB3132	:REAL;	(*	HUS2_FA203_FF01_RMAN	AS01	GVL.HUS2_FA203_FF01_RMAN	REAL	0	100	0	100	%		Manuell styrsignal frånluftsfläkt			*)
																			
		HUS2_FA203_GT51_STAG	AT%MB3136	:REAL;	(*	HUS2_FA203_GT51_STAG	AS01	GVL.HUS2_FA203_GT51_STAG	REAL	0	50	0	50	°C	0.0	Gränsvärde start forcering frånluftsfläkt			*)
		HUS2_FA203_GT51_STOG	AT%MB3140	:REAL;	(*	HUS2_FA203_GT51_STOG	AS01	GVL.HUS2_FA203_GT51_STOG	REAL	0	50	0	50	°C	0.0	Gränsvärde stopp forcering frånluftsfläkt			*)
																			
		HUS2_FA203_GT51_GVH	AT%MB3144	:REAL;	(*	HUS2_FA203_GT51_GVH	AS01	GVL.HUS2_FA203_GT51_GVH	REAL	0	50	0	50	°C	0.0	Gränsvärde hög temperatur			*)
		HUS2_FA203_GT51_FLG	AT%MB3148	:INT;	(*	HUS2_FA203_GT51_FLG	AS01	GVL.HUS2_FA203_GT51_FLG	INT	0	3600	0	3600	Min		Lamfördröjning hög temperatur			*)
																			

		HUS2_FA203_GT51_KRV	AT%MB3156	:REAL;	(*	HUS2_FA203_GT51_KRV	AS01	GVL.HUS2_FA203_GT51_KRV	REAL	-10	10	-10	10	°C	0.0	Kalibreringsvärde frånluftsgivare			*)
																			
		HUS2_FA203_FF01_BV	AT%MB3160	:REAL;	(*	HUS2_FA203_FF01_BV	AS01	GVL.HUS2_FA203_FF01_BV	REAL	0	100	0	100	%		Grundflöde frånluftsfläkt			*)
		HUS2_FA203_FF01_BV1	AT%MB3164	:REAL;	(*	HUS2_FA203_FF01_BV1	AS01	GVL.HUS2_FA203_FF01_BV1	REAL	0	100	0	100	%		Forcerat flöde frånluftsfläkt			*)
																			
																			
																			
																			
																			
																			


END_VAR
																
																

(* Global variable list: HUS2/FA201, FA202, FA203/HUS2_FA201_203_LARM *)
VAR_GLOBAL



																								
																								
	HUS2_FA201_SO1_LM	AT%MX3200.0	:BOOL; 	(*	HUS2_FA201_SO1_LM	AS01	GVL.HUS2_FA201_SO1_LM	DIGITAL	0	0	0	0			Serviceomkopplare ej i läge AUTO	p:C		*)						
	HUS2_FA201_FF01_LM	AT%MX3200.1	:BOOL; 	(*	HUS2_FA201_FF01_LM	AS01	GVL.HUS2_FA201_FF01_LM	DIGITAL	0	0	0	0			Frånluftsfläkt ej i AUTO	p:B		*)						
	HUS2_FA201_GT51_LG	AT%MX3200.2	:BOOL; 	(*	HUS2_FA201_GT51_LG	AS01	GVL.HUS2_FA201_GT51_LG	DIGITAL	0	0	0	0			Givarfel frånluftsgivare	p:B		*)						
	HUS2_FA201_GT51_LH	AT%MX3200.3	:BOOL; 	(*	HUS2_FA201_GT51_LH	AS01	GVL.HUS2_FA201_GT51_LH	DIGITAL	0	0	0	0			Hög temperatur	p:B		*)						
																								
	HUS2_FA201_FF01_ACK	AT%MX3201.0	:BOOL; 	(*	HUS2_FA201_FF01_ACK	AS01	GVL.HUS2_FA201_FF01_ACK	DIGITAL	0	0	0	0			Larmkvittens frånluftsfläkt			*)						
																								
																								
	HUS2_FA202_SO1_LM	AT%MX3202.0	:BOOL; 	(*	HUS2_FA202_SO1_LM	AS01	GVL.HUS2_FA202_SO1_LM	DIGITAL	0	0	0	0			Serviceomkopplare ej i läge AUTO	p:C		*)						
	HUS2_FA202_FF01_LM	AT%MX3202.1	:BOOL; 	(*	HUS2_FA202_FF01_LM	AS01	GVL.HUS2_FA202_FF01_LM	DIGITAL	0	0	0	0			Frånluftsfläkt ej i AUTO	p:B		*)						
	HUS2_FA202_GT51_LG	AT%MX3202.2	:BOOL; 	(*	HUS2_FA202_GT51_LG	AS01	GVL.HUS2_FA202_GT51_LG	DIGITAL	0	0	0	0			Givarfel frånluftsgivare	p:B		*)						
	HUS2_FA202_GT51_LH	AT%MX3202.3	:BOOL; 	(*	HUS2_FA202_GT51_LH	AS01	GVL.HUS2_FA202_GT51_LH	DIGITAL	0	0	0	0			Hög temperatur	p:B		*)						
																								
	HUS2_FA202_FF01_ACK	AT%MX3203.0	:BOOL; 	(*	HUS2_FA202_FF01_ACK	AS01	GVL.HUS2_FA202_FF01_ACK	DIGITAL	0	0	0	0			Larmkvittens frånluftsfläkt			*)						
																								
																								
	HUS2_FA203_SO1_LM	AT%MX3204.0	:BOOL; 	(*	HUS2_FA203_SO1_LM	AS01	GVL.HUS2_FA203_SO1_LM	DIGITAL	0	0	0	0			Serviceomkopplare ej i läge AUTO	p:C		*)						
	HUS2_FA203_FF01_LM	AT%MX3204.1	:BOOL; 	(*	HUS2_FA203_FF01_LM	AS01	GVL.HUS2_FA203_FF01_LM	DIGITAL	0	0	0	0			Frånluftsfläkt ej i AUTO	p:B		*)						
	HUS2_FA203_GT51_LG	AT%MX3204.2	:BOOL; 	(*	HUS2_FA203_GT51_LG	AS01	GVL.HUS2_FA203_GT51_LG	DIGITAL	0	0	0	0			Givarfel frånluftsgivare	p:B		*)						
	HUS2_FA203_GT51_LH	AT%MX3204.3	:BOOL; 	(*	HUS2_FA203_GT51_LH	AS01	GVL.HUS2_FA203_GT51_LH	DIGITAL	0	0	0	0			Hög temperatur	p:B		*)						
																								
	HUS2_FA203_FF01_ACK	AT%MX3205.0	:BOOL; 	(*	HUS2_FA203_FF01_ACK	AS01	GVL.HUS2_FA203_FF01_ACK	DIGITAL	0	0	0	0			Larmkvittens frånluftsfläkt			*)						
																								
																								
																								
																								
																								

																								


END_VAR

(* Global variable list: HUS2/FA201, FA202, FA203/HUS2_FA201_203_OVRIGT *)
VAR_GLOBAL

																						
	HUS2_FA201_SO1_IH	AT%MX3210.0	:BOOL;	(*	HUS2_FA201_SO1_IH	AS01	GVL.HUS2_FA201_SO1_IH	DIGITAL	0	0	0	0			Serviceomkopplare ej i AUTO			*)				
	HUS2_FA201_SO1_IA	AT%MX3210.1	:BOOL;	(*	HUS2_FA201_SO1_IA	AS01	GVL.HUS2_FA201_SO1_IA	DIGITAL	0	0	0	0			Serviceomkopplare i läge AUTO			*)				
	HUS2_FA201_SO1_IF	AT%MX3210.2	:BOOL;	(*	HUS2_FA201_SO1_IF	AS01	GVL.HUS2_FA201_SO1_IF	DIGITAL	0	0	0	0			Serviceomkopplare i läge 0			*)				
	HUS2_FA201_SO1_IT	AT%MX3210.3	:BOOL;	(*	HUS2_FA201_SO1_IT	AS01	GVL.HUS2_FA201_SO1_IT	DIGITAL	0	0	0	0			Serviceomkopplare i läge HAND TILL			*)				

	HUS2_FA201_FF01_IT	AT%MX3210.5	:BOOL;	(*	HUS2_FA201_FF01_IT	AS01	GVL.HUS2_FA201_FF01_IT	DIGITAL	0	0	0	0			Frånluftsfläkt indikering TILL			*)				
																						
																						
	HUS2_FA202_SO1_IH	AT%MX3211.0	:BOOL;	(*	HUS2_FA202_SO1_IH	AS01	GVL.HUS2_FA202_SO1_IH	DIGITAL	0	0	0	0			Serviceomkopplare ej i AUTO			*)				
	HUS2_FA202_SO1_IA	AT%MX3211.1	:BOOL;	(*	HUS2_FA202_SO1_IA	AS01	GVL.HUS2_FA202_SO1_IA	DIGITAL	0	0	0	0			Serviceomkopplare i läge AUTO			*)				
	HUS2_FA202_SO1_IF	AT%MX3211.2	:BOOL;	(*	HUS2_FA202_SO1_IF	AS01	GVL.HUS2_FA202_SO1_IF	DIGITAL	0	0	0	0			Serviceomkopplare i läge 0			*)				
	HUS2_FA202_SO1_IT	AT%MX3211.3	:BOOL;	(*	HUS2_FA202_SO1_IT	AS01	GVL.HUS2_FA202_SO1_IT	DIGITAL	0	0	0	0			Serviceomkopplare i läge HAND TILL			*)				

	HUS2_FA202_FF01_IT	AT%MX3211.5	:BOOL;	(*	HUS2_FA202_FF01_IT	AS01	GVL.HUS2_FA202_FF01_IT	DIGITAL	0	0	0	0			Frånluftsfläkt indikering TILL			*)				
																						
																						
	HUS2_FA203_SO1_IH	AT%MX3212.0	:BOOL;	(*	HUS2_FA203_SO1_IH	AS01	GVL.HUS2_FA203_SO1_IH	DIGITAL	0	0	0	0			Serviceomkopplare ej i AUTO			*)				
	HUS2_FA203_SO1_IA	AT%MX3212.1	:BOOL;	(*	HUS2_FA203_SO1_IA	AS01	GVL.HUS2_FA203_SO1_IA	DIGITAL	0	0	0	0			Serviceomkopplare i läge AUTO			*)				
	HUS2_FA203_SO1_IF	AT%MX3212.2	:BOOL;	(*	HUS2_FA203_SO1_IF	AS01	GVL.HUS2_FA203_SO1_IF	DIGITAL	0	0	0	0			Serviceomkopplare i läge 0			*)				
	HUS2_FA203_SO1_IT	AT%MX3212.3	:BOOL;	(*	HUS2_FA203_SO1_IT	AS01	GVL.HUS2_FA203_SO1_IT	DIGITAL	0	0	0	0			Serviceomkopplare i läge HAND TILL			*)				

	HUS2_FA203_FF01_IT	AT%MX3212.5	:BOOL;	(*	HUS2_FA203_FF01_IT	AS01	GVL.HUS2_FA203_FF01_IT	DIGITAL	0	0	0	0			Frånluftsfläkt indikering TILL			*)				
																						
																						



END_VAR

(* Global variable list: HUS2/VS1 & VP1/HUS2_VS1_INST *)
VAR_GLOBAL PERSISTENT




				(*	Name	Device	Address	Data type	Rawmin	Rawmax	Engmin	Engmax	Unit	Format	Description	Alarmoptions	Trendoptions	*)	
																			
	HUS2_VS1_GT11_UX1	AT%MB2000	:REAL;	(*	HUS2_VS1_GT11_UX1	AS01	GVL.HUS2_VS1_GT11_UX1	REAL	-50	150	-50	150	°C	3.1 EU	Utetemp. kompenserad kurva Brytpunkt X1			*)	
	HUS2_VS1_GT11_UX2	AT%MB2004	:REAL;	(*	HUS2_VS1_GT11_UX2	AS01	GVL.HUS2_VS1_GT11_UX2	REAL	-50	150	-50	150	°C	3.1 EU	Utetemp. kompenserad kurva Brytpunkt X2			*)	
	HUS2_VS1_GT11_UX3	AT%MB2008	:REAL;	(*	HUS2_VS1_GT11_UX3	AS01	GVL.HUS2_VS1_GT11_UX3	REAL	-50	150	-50	150	°C	3.1 EU	Utetemp. kompenserad kurva Brytpunkt X3			*)	
	HUS2_VS1_GT11_UX4	AT%MB2012	:REAL;	(*	HUS2_VS1_GT11_UX4	AS01	GVL.HUS2_VS1_GT11_UX4	REAL	-50	150	-50	150	°C	3.1 EU	Utetemp. kompenserad kurva Brytpunkt X4			*)	
	HUS2_VS1_GT11_UX5	AT%MB2016	:REAL;	(*	HUS2_VS1_GT11_UX5	AS01	GVL.HUS2_VS1_GT11_UX5	REAL	-50	150	-50	150	°C	3.1 EU	Utetemp. kompenserad kurva Brytpunkt X5			*)	
	HUS2_VS1_GT11_UY1	AT%MB2020	:REAL;	(*	HUS2_VS1_GT11_UY1	AS01	GVL.HUS2_VS1_GT11_UY1	REAL	-50	150	-50	150	°C	3.1 EU	Utetemp. kompenserad kurva Brytpunkt Y1			*)	
	HUS2_VS1_GT11_UY2	AT%MB2024	:REAL;	(*	HUS2_VS1_GT11_UY2	AS01	GVL.HUS2_VS1_GT11_UY2	REAL	-50	150	-50	150	°C	3.1 EU	Utetemp. kompenserad kurva Brytpunkt Y2			*)	
	HUS2_VS1_GT11_UY3	AT%MB2028	:REAL;	(*	HUS2_VS1_GT11_UY3	AS01	GVL.HUS2_VS1_GT11_UY3	REAL	-50	150	-50	150	°C	3.1 EU	Utetemp. kompenserad kurva Brytpunkt Y3			*)	
	HUS2_VS1_GT11_UY4	AT%MB2032	:REAL;	(*	HUS2_VS1_GT11_UY4	AS01	GVL.HUS2_VS1_GT11_UY4	REAL	-50	150	-50	150	°C	3.1 EU	Utetemp. kompenserad kurva Brytpunkt Y4			*)	
	HUS2_VS1_GT11_UY5	AT%MB2036	:REAL;	(*	HUS2_VS1_GT11_UY5	AS01	GVL.HUS2_VS1_GT11_UY5	REAL	-50	150	-50	150	°C	3.1 EU	Utetemp. kompenserad kurva Brytpunkt Y5			*)	
	HUS2_VS1_GT11_UMIN	AT%MB2040	:REAL;	(*	HUS2_VS1_GT11_UMIN	AS01	GVL.HUS2_VS1_GT11_UMIN	REAL	-50	150	-50	150	°C	3.1 EU	Utetemp. kompenserad kurva Min-begränsning			*)	
	HUS2_VS1_GT11_UMAX	AT%MB2044	:REAL;	(*	HUS2_VS1_GT11_UMAX	AS01	GVL.HUS2_VS1_GT11_UMAX	REAL	-50	150	-50	150	°C	3.1 EU	Utetemp. kompenserad kurva Max-begränsning			*)	
																			
		HUS2_VS1_GT11_CP	AT%MB2048	:REAL;	(*	HUS2_VS1_GT11_CPV	AS01	GVL.HUS2_VS1_GT11_CP	REAL	0	10	0	10		0.0	P-parameter			*)
		HUS2_VS1_GT11_CI	AT%MB2052	:REAL;	(*	HUS2_VS1_GT11_CIV	AS01	GVL.HUS2_VS1_GT11_CI	REAL	0	900	0	900	Sek		I-Tid 			*)
		HUS2_VS1_GT11_CD	AT%MB2056	:REAL;	(*	HUS2_VS1_GT11_CDV	AS01	GVL.HUS2_VS1_GT11_CD	REAL	0	900	0	900	Sek		D-tid 			*)
		HUS2_VS1_GT11_CS	AT%MB2060	:REAL;	(*	HUS2_VS1_GT11_CSV	AS01	GVL.HUS2_VS1_GT11_CS	REAL	0	900	0	900	Sek		Samplingstid			*)	
		HUS2_VS1_GT11_CZ	AT%MB2064	:REAL;	(*	HUS2_VS1_GT11_CZV	AS01	GVL.HUS2_VS1_GT11_CZ	REAL	-10	10	-10	10	°C	0.0	Dödband regulator			*)	
																				
		HUS2_VS1_SO1_MAN	AT%MB2068	:INT;	(*	HUS2_VS1_SO1_MAN	AS01	GVL.HUS2_VS1_SO1_MAN	INT	0	2	0	2			Manuell styrning system VS1. 0=Auto, 1=Manuell från, 2=Manuell till			*)	
		HUS2_VS1_PV01_MAN	AT%MB2070	:INT;	(*	HUS2_VS1_PV01_MAN	AS01	GVL.HUS2_VS1_PV01_MAN	INT	0	2	0	2			Manuell styrning crikulationspump 0=Auto,1=Från,2=Till			*)	
		HUS2_VS1_SV11_MAN1	AT%MB2072	:INT;	(*	HUS2_VS1_SV11_MAN	AS01	GVL.HUS2_VS1_SV11_MAN	INT	0	1	0	1			Manuell styrning ventilställdon 0=Auto,1=Hand			*)	
		HUS2_VS1_SV11_RMAN	AT%MB2076	:REAL;	(*	HUS2_VS1_SV11_RMAN	AS01	GVL.HUS2_VS1_SV11_RMAN	REAL	0	100	0	100	%		Manuell styrsignal ventilställdon			*)	
																				
		HUS2_VS1_SO1_FLM	AT%MB2080	:INT;	(*	HUS2_VS1_SO1_FLM	AS01	GVL.HUS2_VS1_SO1_FLM	INT	0	3600	0	3600	Min		Larmfördröjning serviceomkopplare ej i läge AUTO			*)	
		HUS2_VS1_PV01_FLM	AT%MB2082	:INT;	(*	HUS2_VS1_PV01_FLM	AS01	GVL.HUS2_VS1_PV01_FLM	INT	0	3600	0	3600	Min		Larmfördröjning cirkulationspump ej i AUTO			*)	
		HUS2_VS1_SV11_FLM	AT%MB2084	:INT;	(*	HUS2_VS1_SV11_FLM	AS01	GVL.HUS2_VS1_SV11_FLM	INT	0	3600	0	3600	Min		Larmfördröjning ventilställdon ej i AUTO			*)	
		HUS2_VS1_PV01_FLD	AT%MB2086	:INT;	(*	HUS2_VS1_PV01_FLD	AS01	GVL.HUS2_VS1_PV01_FLD	INT	0	120	0	120	Sek		Larmfördröjning driftfel cirkulationspump			*)	
																				
		HUS2_VS1_GT11_GAVH	AT%MB2088	:REAL;	(*	HUS2_VS1_GT11_GAVH	AS01	GVL.HUS2_VS1_GT11_GAVH	REAL	-20	20	-20	20	°C	0.0	Gränsavvikelse hög framledningstemperatur			*)	
		HUS2_VS1_GT11_GAVL	AT%MB2092	:REAL;	(*	HUS2_VS1_GT11_GAVL	AS01	GVL.HUS2_VS1_GT11_GAVL	REAL	-20	20	-20	20	°C	0.0	Gränsavvikelse låg framledningstemperatur			*)
		HUS2_VS1_GT11_FLAH	AT%MB2096	:INT;	(*	HUS2_VS1_GT11_FLAH	AS01	GVL.HUS2_VS1_GT11_FLAH	INT	0	3600	0	3600	Min		Larmfördröjning hög framledningstemperatur			*)	
		HUS2_VS1_GT11_FLAL	AT%MB2098	:INT;	(*	HUS2_VS1_GT11_FLAL	AS01	GVL.HUS2_VS1_GT11_FLAL	INT	0	3600	0	3600	Min		Lamfördröjning låg framledningstemperatur			*)	
																				
		HUS2_VS1_GP41_GVL	AT%MB2100	:REAL;	(*	HUS2_VS1_GP41_GVL	AS01	GVL.HUS2_VS1_GP41_GVL	REAL	0	20	0	20	Bar		Gränsvärde lågt systemtryck			*)	
		HUS2_VS1_GP41_GVH	AT%MB2104	:REAL;	(*	HUS2_VS1_GP41_GVH	AS01	GVL.HUS2_VS1_GP41_GVH	REAL	0	20	0	20	Bar		Gränsvärde högt systemtryck			*)	
		HUS2_VS1_GP41_FLGH	AT%MB2108	:INT;	(*	HUS2_VS1_GP41_FLGH	AS01	GVL.HUS2_VS1_GP41_FLGH	INT	0	3600	0	3600	Min		Larmfördröjning lågt systemtryck			*)	
		HUS2_VS1_GP41_FLGL	AT%MB2110	:INT;	(*	HUS2_VS1_GP41_FLGL	AS01	GVL.HUS2_VS1_GP41_FLGL	INT	0	3600	0	3600	Min		Larmfördröjning högt systemtryck			*)	

		HUS2_VS1_GT11_KRV	AT%MB2116	:REAL;	(*	HUS2_VS1_GT11_KRV	AS01	GVL.HUS2_VS1_GT11_KRV	REAL	-10	10	-10	10	°C	0.0	Kalibreringsvärde framledningsgivare			*)	
		HUS2_VS1_GT41_KRV	AT%MB2120	:REAL;	(*	HUS2_VS1_GT41_KRV	AS01	GVL.HUS2_VS1_GT41_KRV	REAL	-10	10	-10	10	°C	0.0	Kalibreringsvärde returgivare			*)	

																				
		HUS2_VP1_TK01_HHMM	AT%MB2124	:INT;	(*	HUS2_VP1_TK01_HHMM	AS01	GVL.HUS2_VP1_TK01_HHMM	INT	0	2359	0	2359	HHMM		Starttid  läckagekontroll VP1 HHMM			*)	
		HUS2_VP1_TK01_HHMM1	AT%MB2126	:INT;	(*	HUS2_VP1_TK01_HHMM1	AS01	GVL.HUS2_VP1_TK01_HHMM1	INT	0	2359	0	2359	HHMM		Stopptid läckagekontroll VP1 HHMM			*)	
		HUS2_VP1_TK01_VDAG	AT%MB2128	:INT;	(*	HUS2_VP1_TK01_VDAG	AS01	GVL.HUS2_VP1_TK01_VDAG	INT	0	6	0	6	Veckodag		Veckodag för läckagekontroll VP1 (0=Sön..6=Lör)			*)	
		HUS2_VP1_TK01_MAN	AT%MB2130	:INT;	(*	HUS2_VP1_TK01_MAN	AS01	GVL.HUS2_VP1_TK01_MAN	INT	0	2	0	2			Manuell styrning läckagekontroll VP1 0=Auto, 1=Manuell från, 2=Manuell till			*)	
		HUS2_VP1_TK01_FLM	AT%MB2132	:INT;	(*	HUS2_VP1_TK01_FLM	AS01	GVL.HUS2_VP1_TK01_FLM	INT	0	3600	0	3600	Min		Larmfördröjning läckagekontroll VP1 ej i AUTO			*)	
																				
		HUS2_VP1_MQ41_UX1	AT%MB2136	:REAL;	(*	HUS2_VP1_MQ41_UX1	AS01	GVL.HUS2_VP1_MQ41_UX1	REAL	-50	150	-50	150	°C	0.0	Utetemp. kompenserad kurva Brytpunkt X1			*)	
		HUS2_VP1_MQ41_UX2	AT%MB2140	:REAL;	(*	HUS2_VP1_MQ41_UX2	AS01	GVL.HUS2_VP1_MQ41_UX2	REAL	-50	150	-50	150	°C	0.0	Utetemp. kompenserad kurva Brytpunkt X2			*)	
		HUS2_VP1_MQ41_UX3	AT%MB2144	:REAL;	(*	HUS2_VP1_MQ41_UX3	AS01	GVL.HUS2_VP1_MQ41_UX3	REAL	-50	150	-50	150	°C	0.0	Utetemp. kompenserad kurva Brytpunkt X3			*)	
		HUS2_VP1_MQ41_UX4	AT%MB2148	:REAL;	(*	HUS2_VP1_MQ41_UX4	AS01	GVL.HUS2_VP1_MQ41_UX4	REAL	-50	150	-50	150	°C	0.0	Utetemp. kompenserad kurva Brytpunkt X4			*)	
		HUS2_VP1_MQ41_UX5	AT%MB2152	:REAL;	(*	HUS2_VP1_MQ41_UX5	AS01	GVL.HUS2_VP1_MQ41_UX5	REAL	-50	150	-50	150	°C	0.0	Utetemp. kompenserad kurva Brytpunkt X5			*)	
		HUS2_VP1_MQ41_UY1	AT%MB2156	:REAL;	(*	HUS2_VP1_MQ41_UY1	AS01	GVL.HUS2_VP1_MQ41_UY1	REAL	0	500	0	500	kWh	0.0	Utetemp. kompenserad kurva Brytpunkt Y1			*)	
		HUS2_VP1_MQ41_UY2	AT%MB2160	:REAL;	(*	HUS2_VP1_MQ41_UY2	AS01	GVL.HUS2_VP1_MQ41_UY2	REAL	0	500	0	500	kWh	0.0	Utetemp. kompenserad kurva Brytpunkt Y2			*)	
		HUS2_VP1_MQ41_UY3	AT%MB2164	:REAL;	(*	HUS2_VP1_MQ41_UY3	AS01	GVL.HUS2_VP1_MQ41_UY3	REAL	0	500	0	500	kWh	0.0	Utetemp. kompenserad kurva Brytpunkt Y3			*)	
		HUS2_VP1_MQ41_UY4	AT%MB2168	:REAL;	(*	HUS2_VP1_MQ41_UY4	AS01	GVL.HUS2_VP1_MQ41_UY4	REAL	0	500	0	500	kWh	0.0	Utetemp. kompenserad kurva Brytpunkt Y4			*)	
		HUS2_VP1_MQ41_UY5	AT%MB2172	:REAL;	(*	HUS2_VP1_MQ41_UY5	AS01	GVL.HUS2_VP1_MQ41_UY5	REAL	0	500	0	500	kWh	0.0	Utetemp. kompenserad kurva Brytpunkt Y5			*)	
		HUS2_VP1_MQ41_UMIN	AT%MB2176	:REAL;	(*	HUS2_VP1_MQ41_UMIN	AS01	GVL.HUS2_VP1_MQ41_UMIN	REAL	0	500	0	500	kWh	0.0	Utetemp. kompenserad kurva Min-begränsning			*)	
		HUS2_VP1_MQ41_UMAX	AT%MB2180	:REAL;	(*	HUS2_VP1_MQ41_UMAX	AS01	GVL.HUS2_VP1_MQ41_UMAX	REAL	0	500	0	500	kWh	0.0	Utetemp. kompenserad kurva Max-begränsning			*)	

		HUS2_VP1_MQ41_CP	AT%MB2184	:REAL;	(*	HUS2_VP1_MQ41_CP	AS01	GVL.HUS2_VP1_MQ41_CP	REAL	0	10	0	10		0.0	P-parameter			*)	
		HUS2_VP1_MQ41_CI	AT%MB2188	:REAL;	(*	HUS2_VP1_MQ41_CI	AS01	GVL.HUS2_VP1_MQ41_CI	REAL	0	900	0	900	Sek		I-Tid 			*)
		HUS2_VP1_MQ41_CD	AT%MB2192	:REAL;	(*	HUS2_VP1_MQ41_CD	AS01	GVL.HUS2_VP1_MQ41_CD	REAL	0	900	0	900	Sek		D-tid 			*)
		HUS2_VP1_MQ41_CS	AT%MB2196	:REAL;	(*	HUS2_VP1_MQ41_CS	AS01	GVL.HUS2_VP1_MQ41_CS	REAL	0	900	0	900	Sek		Samplingstid			*)	
		HUS2_VP1_MQ41_CZ	AT%MB2200	:REAL;	(*	HUS2_VP1_MQ41_CZ	AS01	GVL.HUS2_VP1_MQ41_CZ	REAL	-10	10	-10	10	°C	0.0	Dödband regulator			*)	
																				
		HUS2_VP1_MQ41_SO1_MAN	AT%MB2204	:INT;	(*	HUS2_VP1_MQ41_SO1_MAN	AS01	GVL.HUS2_VP1_MQ41_SO1_MAN	INT	0	1	0	1			Manuell styrning effektbegränsning VP1 0=Från, 1=Till			*)

																				
																				


	END_VAR
																
																

(* Global variable list: HUS2/VS1 & VP1/HUS2_VS1_LARM *)
VAR_GLOBAL


																								
		HUS2_VS1_SO1_LM	AT%MX2510.0	:BOOL; 	(*	HUS2_VS1_SO1_LM	AS01	GVL.HUS2_VS1_SO1_LM	DIGITAL	0	0	0	0			Serviceomkopplare ej i läge AUTO	p:C		*)					
		HUS2_VS1_PV01_LM	AT%MX2510.1	:BOOL; 	(*	HUS2_VS1_PV01_LM	AS01	GVL.HUS2_VS1_PV01_LM	DIGITAL	0	0	0	0			Cirkulationspump ej i AUTO	p:B		*)					
		HUS2_VS1_SV11_LM	AT%MX2510.2	:BOOL; 	(*	HUS2_VS1_SV11_LM	AS01	GVL.HUS2_VS1_SV11_LM	DIGITAL	0	0	0	0			Ventilställdon ej i AUTO	p:B		*)					
		HUS2_VS1_PV01_LD	AT%MX2510.3	:BOOL; 	(*	HUS2_VS1_PV01_LD	AS01	GVL.HUS2_VS1_PV01_LD	DIGITAL	0	0	0	0			Driftfel cirkulationspump	p:B		*)					
		HUS2_VS1_GT11_LG	AT%MX2510.4	:BOOL; 	(*	HUS2_VS1_GT11_LG	AS01	GVL.HUS2_VS1_GT11_LG	DIGITAL	0	0	0	0			Givarfel framledningsgivare	p:B		*)					
		HUS2_VS1_GT41_LG	AT%MX2510.5	:BOOL; 	(*	HUS2_VS1_GT41_LG	AS01	GVL.HUS2_VS1_GT41_LG	DIGITAL	0	0	0	0			Givarfel returgivare	p:B		*)					
		HUS2_VS1_GT11_LAH	AT%MX2510.6	:BOOL; 	(*	HUS2_VS1_GT11_LAH	AS01	GVL.HUS2_VS1_GT11_LAH	DIGITAL	0	0	0	0			Larmavvikelse hög framledningstemp	p:B		*)					
		HUS2_VS1_GT11_LAL	AT%MX2510.7	:BOOL; 	(*	HUS2_VS1_GT11_LAL	AS01	GVL.HUS2_VS1_GT11_LAL	DIGITAL	0	0	0	0			Larmavvikelse låg framledningstemp	p:B		*)					
		HUS2_VS1_GP41_LL	AT%MX2511.0	:BOOL; 	(*	HUS2_VS1_GP41_LL	AS01	GVL.HUS2_VS1_GP41_LL	DIGITAL	0	0	0	0			Lågt systemtryck	p:A		*)					
		HUS2_VS1_GP41_LH	AT%MX2511.1	:BOOL; 	(*	HUS2_VS1_GP41_LH	AS01	GVL.HUS2_VS1_GP41_LH	DIGITAL	0	0	0	0			Högt systemtryck	p:A		*)
		HUS2_VP1_MQ41_L	AT%MX2511.2	:BOOL; 	(*	HUS2_VP1_MQ41_L	AS01	GVL.HUS2_VP1_MQ41_L	DIGITAL	0	0	0	0			Summalarm energimätare	p:B		*)
		HUS2_VP1_MQ41_LC	AT%MX2511.3	:BOOL; 	(*	HUS2_VP1_MQ41_LC	AS01	GVL.HUS2_VP1_MQ41_LC	DIGITAL	0	0	0	0			Kommunikationsfel energimätare	p:B		*)					
		HUS2_VP1_L	AT%MX2511.4	:BOOL; 	(*	HUS2_VP1_L	AS01	GVL.HUS2_VP1_L	DIGITAL	0	0	0	0			Läckagelarm	p:B		*)
		HUS2_VP1_TK01_LM	AT%MX2511.5	:BOOL;	(*	HUS2_VP1_TK01_LM	AS01	GVL.HUS2_VP1_TK01_LM	DIGITAL	0	0	0	0			Larm läckagekontroll VP1 ej i AUTO	p:C		*)


																								

																								
																								
		HUS2_VS1_PV01_ACK	AT%MX2518.0	:BOOL; 	(*	HUS2_VS1_PV01_ACK	AS01	GVL.HUS2_VS1_PV01_ACK	DIGITAL	0	0	0	0			Larmkvittens pump			*)					
		HUS2_VP1_ACK	AT%MX2518.1	:BOOL; 	(*	HUS2_VP1_ACK	AS01	GVL.HUS2_VP1_ACK	DIGITAL	0	0	0	0			Larmkvittens läckagelarm			*)

																								
																								

																			
																			



END_VAR

(* Global variable list: HUS2/VS1 & VP1/HUS2_VS1_OVRIGT *)
VAR_GLOBAL




	HUS2_VS1_SO1_IH	AT%MX2520.0	:BOOL;	(*	HUS2_VS1_SO1_IH	AS01	GVL.HUS2_VS1_SO1_IH	DIGITAL	0	0	0	0			Serviceomkopplare ej i AUTO			*)					
	HUS2_VS1_SO1_IA	AT%MX2520.1	:BOOL;	(*	HUS2_VS1_SO1_IA	AS01	GVL.HUS2_VS1_SO1_IA	DIGITAL	0	0	0	0			Serviceomkopplare i läge AUTO			*)					
	HUS2_VS1_SO1_IF	AT%MX2520.2	:BOOL;	(*	HUS2_VS1_SO1_IF	AS01	GVL.HUS2_VS1_SO1_IF	DIGITAL	0	0	0	0			Serviceomkopplare i läge 0			*)					
	HUS2_VS1_SO1_IT	AT%MX2520.3	:BOOL;	(*	HUS2_VS1_SO1_IT	AS01	GVL.HUS2_VS1_SO1_IT	DIGITAL	0	0	0	0			Serviceomkopplare i läge HAND TILL			*)
	HUS2_VP1_TK01_IT	AT%MX2520.5	:BOOL;	(*	HUS2_VP1_TK01_IT	AS01	GVL.HUS2_VP1_TK01_IT	DIGITAL	0	0	0	0			Tidkanal läckagekontroll Aktiv			*)

